C01814=1052.685,226.310,-95.287,172.073,35.922,156.749
C01815=1052.692,226.559,-95.315,172.074,35.926,156.749
C01816=1052.699,226.807,-95.341,172.076,35.929,156.750
C01817=1052.705,227.055,-95.369,172.079,35.932,156.751
C01818=1052.711,227.304,-95.396,172.081,35.936,156.752
C01819=1052.718,227.552,-95.423,172.083,35.939,156.752
C01820=1052.724,227.801,-95.450,172.086,35.942,156.753
C01821=1052.731,228.049,-95.478,172.088,35.946,156.754
C01822=1052.736,228.298,-95.504,172.089,35.950,156.754
C01823=1052.743,228.546,-95.532,172.092,35.953,156.755
C01824=1052.750,228.795,-95.560,172.094,35.956,156.756
C01825=1052.756,229.043,-95.586,172.097,35.960,156.756
C01826=1052.763,229.291,-95.614,172.099,35.963,156.757
C01827=1052.769,229.541,-95.641,172.101,35.966,156.758
C01828=1052.775,229.788,-95.669,172.104,35.970,156.759
C01829=1052.781,230.037,-95.696,172.105,35.974,156.759
C01830=1052.788,230.286,-95.723,172.107,35.977,156.760
C01831=1052.794,230.534,-95.751,172.110,35.980,156.761
C01832=1052.800,230.782,-95.778,172.112,35.984,156.761
C01833=1052.807,231.031,-95.805,172.114,35.987,156.762
C01834=1052.813,231.279,-95.833,172.117,35.990,156.763
C01835=1052.820,231.527,-95.860,172.119,35.994,156.763
C01836=1052.826,231.776,-95.888,172.122,35.997,156.764
C01837=1052.831,232.024,-95.915,172.123,36.001,156.765
C01838=1052.838,232.273,-95.943,172.125,36.004,156.766
C01839=1052.845,232.521,-95.971,172.128,36.008,156.766
C01840=1052.851,232.770,-95.999,172.130,36.011,156.767
C01841=1052.857,233.018,-96.025,172.132,36.015,156.768
C01842=1052.864,233.266,-96.053,172.135,36.018,156.768
C01843=1052.870,233.515,-96.081,172.137,36.021,156.769
C01844=1052.876,233.763,-96.109,172.139,36.025,156.770
C01845=1052.883,234.011,-96.136,172.142,36.028,156.771
C01846=1052.889,234.260,-96.164,172.144,36.031,156.771
C01847=1052.895,234.508,-96.192,172.146,36.035,156.772
C01848=1052.901,234.754,-96.219,172.148,36.039,156.773
C01849=1052.908,235.000,-96.246,172.150,36.042,156.773
C01850=1052.914,235.245,-96.274,172.153,36.045,156.774
C01851=1052.920,235.491,-96.301,172.155,36.049,156.775
C01852=1052.926,235.736,-96.329,172.157,36.052,156.775
C01853=1052.932,235.982,-96.356,172.160,36.055,156.776
C01854=1052.939,236.227,-96.384,172.162,36.059,156.777
C01855=1052.945,236.473,-96.411,172.164,36.062,156.777
C01856=1052.951,236.722,-96.439,172.167,36.065,156.778
C01857=1052.957,236.969,-96.466,172.169,36.069,156.779
C01858=1052.964,237.218,-96.494,172.172,36.072,156.780
C01859=1052.971,237.466,-96.522,172.174,36.076,156.780
C01860=1052.977,237.715,-96.550,172.175,36.079,156.781
C01861=1052.983,237.963,-96.578,172.178,36.082,156.782
C01862=1052.990,238.212,-96.606,172.180,36.086,156.782
C01863=1052.996,238.459,-96.634,172.182,36.089,156.783
C01864=1053.002,238.708,-96.662,172.185,36.093,156.784
C01865=1053.009,238.956,-96.690,172.187,36.096,156.785
C01866=1053.015,239.205,-96.718,172.190,36.099,156.785
C01867=1053.022,239.453,-96.746,172.192,36.103,156.786
C01868=1053.028,239.702,-96.774,172.194,36.106,156.787
C01869=1053.034,239.950,-96.802,172.197,36.109,156.787
C01870=1053.040,240.198,-96.829,172.199,36.113,156.788
C01871=1053.047,240.447,-96.857,172.201,36.116,156.789
C01872=1053.053,240.695,-96.886,172.204,36.120,156.789
C01873=1053.060,240.943,-96.914,172.206,36.123,156.790
C01874=1053.067,241.192,-96.941,172.209,36.126,156.791
C01875=1053.072,241.440,-96.970,172.211,36.130,156.792
C01876=1053.079,241.689,-96.998,172.213,36.133,156.792
C01877=1053.085,241.936,-97.026,172.216,36.136,156.793
C01878=1053.091,242.185,-97.054,172.218,36.140,156.794
C01879=1053.097,242.433,-97.082,172.221,36.143,156.794
C01880=1053.104,242.682,-97.110,172.223,36.147,156.795
C01881=1053.110,242.930,-97.139,172.225,36.150,156.796
C01882=1053.116,243.179,-97.167,172.228,36.154,156.797
C01883=1053.123,243.427,-97.195,172.230,36.157,156.797
C01884=1053.129,243.675,-97.224,172.232,36.161,156.798
C01885=1053.135,243.923,-97.252,172.235,36.164,156.799
C01886=1053.142,244.171,-97.281,172.237,36.167,156.799
C01887=1053.148,244.420,-97.309,172.240,36.171,156.800
C01888=1053.154,244.668,-97.337,172.242,36.174,156.801
C01889=1053.160,244.917,-97.366,172.244,36.177,156.802
C01890=1053.167,245.165,-97.393,172.247,36.181,156.802
C01891=1053.173,245.413,-97.422,172.249,36.184,156.803
C01892=1053.179,245.662,-97.451,172.252,36.187,156.804
C01893=1053.186,245.910,-97.478,172.254,36.191,156.804
C01894=1053.192,246.158,-97.508,172.257,36.195,156.805
C01895=1053.198,246.407,-97.536,172.260,36.198,156.806
C01896=1053.204,246.655,-97.565,172.262,36.202,156.807
C01897=1053.211,246.903,-97.593,172.264,36.205,156.807
C01898=1053.217,247.151,-97.621,172.267,36.208,156.808
C01899=1053.223,247.399,-97.650,172.269,36.212,156.809
C01900=1053.229,247.648,-97.679,172.272,36.215,156.809
C01901=1053.235,247.896,-97.708,172.274,36.219,156.810
C01902=1053.241,248.145,-97.736,172.276,36.222,156.811
C01903=1053.248,248.393,-97.764,172.279,36.225,156.812
C01904=1053.254,248.636,-97.793,172.281,36.229,156.812
C01905=1053.260,248.878,-97.820,172.284,36.232,156.813
C01906=1053.266,249.121,-97.849,172.286,36.235,156.814
C01907=1053.272,249.363,-97.877,172.288,36.239,156.814
C01908=1053.279,249.606,-97.905,172.291,36.242,156.815
C01909=1053.284,249.848,-97.933,172.293,36.245,156.816
C01910=1053.290,250.091,-97.961,172.296,36.249,156.817
C01911=1053.297,250.333,-97.989,172.298,36.252,156.817
C01912=1053.303,250.582,-98.018,172.300,36.256,156.818
C01913=1053.310,250.830,-98.047,172.303,36.259,156.819
C01914=1053.316,251.078,-98.075,172.305,36.263,156.819
C01915=1053.322,251.327,-98.104,172.308,36.266,156.820
C01916=1053.328,251.575,-98.133,172.311,36.269,156.821
C01917=1053.334,251.823,-98.163,172.313,36.273,156.822
C01918=1053.340,252.072,-98.191,172.316,36.276,156.822
C01919=1053.347,252.319,-98.219,172.318,36.280,156.823
C01920=1053.354,252.568,-98.248,172.321,36.283,156.824
C01921=1053.360,252.816,-98.277,172.323,36.286,156.824
C01922=1053.366,253.064,-98.306,172.325,36.290,156.825
C01923=1053.372,253.312,-98.335,172.328,36.293,156.826
C01924=1053.378,253.561,-98.364,172.330,36.296,156.827
C01925=1053.385,253.809,-98.393,172.334,36.300,156.827
C01926=1053.391,254.057,-98.422,172.336,36.304,156.828
C01927=1053.398,254.306,-98.451,172.338,36.306,156.829
C01928=1053.404,254.554,-98.480,172.341,36.310,156.829
C01929=1053.411,254.802,-98.509,172.343,36.314,156.830
C01930=1053.417,255.050,-98.538,172.346,36.317,156.831
C01931=1053.423,255.298,-98.567,172.348,36.320,156.832
C01932=1053.430,255.546,-98.596,172.351,36.324,156.832
C01933=1053.436,255.794,-98.625,172.354,36.327,156.833
C01934=1053.443,256.043,-98.654,172.356,36.330,156.834
C01935=1053.449,256.291,-98.683,172.359,36.334,156.834
C01936=1053.455,256.539,-98.712,172.361,36.337,156.835
C01937=1053.461,256.788,-98.741,172.364,36.341,156.836
C01938=1053.468,257.036,-98.770,172.367,36.344,156.837
C01939=1053.475,257.284,-98.800,172.369,36.347,156.837
C01940=1053.481,257.533,-98.829,172.372,36.351,156.838
C01941=1053.487,257.781,-98.858,172.374,36.354,156.839
C01942=1053.493,258.029,-98.887,172.377,36.357,156.839
C01943=1053.500,258.277,-98.915,172.380,36.361,156.840
C01944=1053.507,258.526,-98.945,172.382,36.364,156.841
C01945=1053.513,258.774,-98.974,172.385,36.367,156.842
C01946=1053.520,259.022,-99.003,172.387,36.371,156.842
C01947=1053.526,259.269,-99.033,172.390,36.374,156.843
C01948=1053.533,259.518,-99.062,172.393,36.377,156.844
C01949=1053.539,259.766,-99.091,172.395,36.381,156.844
C01950=1053.546,260.014,-99.120,172.398,36.384,156.845
C01951=1053.552,260.263,-99.149,172.400,36.387,156.846
C01952=1053.559,260.511,-99.179,172.404,36.391,156.847
C01953=1053.565,260.759,-99.208,172.406,36.394,156.847
C01954=1053.571,261.007,-99.237,172.408,36.397,156.848
C01955=1053.578,261.256,-99.267,172.411,36.401,156.849
C01956=1053.585,261.504,-99.296,172.414,36.404,156.849
C01957=1053.591,261.751,-99.326,172.417,36.407,156.850
C01958=1053.598,262.000,-99.355,172.419,36.411,156.851
C01959=1053.604,262.248,-99.384,172.422,36.414,156.852
C01960=1053.610,262.490,-99.413,172.424,36.417,156.852
C01961=1053.617,262.732,-99.442,172.427,36.421,156.853
C01962=1053.623,262.973,-99.470,172.430,36.424,156.854
C01963=1053.629,263.215,-99.499,172.432,36.427,156.854
C01964=1053.635,263.457,-99.528,172.435,36.430,156.855
C01965=1053.642,263.699,-99.557,172.437,36.434,156.856
C01966=1053.648,263.940,-99.585,172.440,36.437,156.856
C01967=1053.654,264.181,-99.614,172.443,36.440,156.857
C01968=1053.660,264.429,-99.644,172.445,36.444,156.858
C01969=1053.667,264.678,-99.674,172.448,36.447,156.859
C01970=1053.674,264.925,-99.703,172.451,36.451,156.859
C01971=1053.679,265.174,-99.733,172.454,36.454,156.860
C01972=1053.686,265.422,-99.763,172.456,36.458,156.861
C01973=1053.692,265.670,-99.792,172.458,36.461,156.862
C01974=1053.698,265.918,-99.823,172.462,36.464,156.862
C01975=1053.705,266.167,-99.852,172.464,36.468,156.863
C01976=1053.712,266.414,-99.882,172.467,36.472,156.864
C01977=1053.717,266.662,-99.912,172.469,36.475,156.865
C01978=1053.724,266.911,-99.941,172.473,36.478,156.865
C01979=1053.731,267.159,-99.971,172.475,36.482,156.866
C01980=1053.736,267.407,-100.001,172.477,36.485,156.867
C01981=1053.744,267.655,-100.031,172.481,36.489,156.867
C01982=1053.750,267.903,-100.061,172.483,36.492,156.868
C01983=1053.756,268.152,-100.091,172.486,36.495,156.869
C01984=1053.763,268.399,-100.121,172.489,36.499,156.870
C01985=1053.769,268.647,-100.151,172.492,36.502,156.870
C01986=1053.775,268.896,-100.180,172.494,36.506,156.871
C01987=1053.781,269.144,-100.211,172.498,36.509,156.872
C01988=1053.788,269.392,-100.241,172.500,36.513,156.873
C01989=1053.794,269.640,-100.271,172.502,36.516,156.873
C01990=1053.801,269.889,-100.301,172.505,36.519,156.874
C01991=1053.807,270.137,-100.331,172.508,36.523,156.875
C01992=1053.813,270.384,-100.361,172.511,36.526,156.876
C01993=1053.820,270.633,-100.391,172.513,36.530,156.876
C01994=1053.826,270.880,-100.421,172.517,36.533,156.877
C01995=1053.833,271.129,-100.452,172.519,36.537,156.878
C01996=1053.839,271.377,-100.481,172.522,36.540,156.879
C01997=1053.846,271.625,-100.512,172.525,36.543,156.879
C01998=1053.852,271.873,-100.541,172.527,36.547,156.880
C01999=1053.858,272.121,-100.572,172.531,36.550,156.881
C02000=1053.865,272.369,-100.602,172.533,36.554,156.882
C02001=1053.871,272.617,-100.633,172.536,36.557,156.882
C02002=1053.877,272.865,-100.663,172.539,36.561,156.883
C02003=1053.884,273.113,-100.693,172.542,36.564,156.884
C02004=1053.890,273.361,-100.723,172.544,36.568,156.885
C02005=1053.897,273.610,-100.754,172.548,36.571,156.885
C02006=1053.903,273.857,-100.784,172.550,36.575,156.886
C02007=1053.910,274.106,-100.815,172.552,36.578,156.887
C02008=1053.915,274.354,-100.845,172.556,36.581,156.887
C02009=1053.923,274.602,-100.875,172.558,36.585,156.888
C02010=1053.928,274.850,-100.905,172.562,36.588,156.889
C02011=1053.935,275.098,-100.936,172.564,36.592,156.890
C02012=1053.941,275.346,-100.966,172.567,36.595,156.891
C02013=1053.948,275.594,-100.997,172.570,36.599,156.891
C02014=1053.954,275.842,-101.027,172.573,36.602,156.892
C02015=1053.960,276.091,-101.058,172.575,36.606,156.893
C02016=1053.966,276.334,-101.088,172.579,36.609,156.894
C02017=1053.973,276.577,-101.118,172.581,36.613,156.894
C02018=1053.979,276.821,-101.148,172.584,36.616,156.895
C02019=1053.985,277.064,-101.178,172.587,36.619,156.896
C02020=1053.992,277.308,-101.208,172.589,36.623,156.896
C02021=1053.999,277.552,-101.238,172.593,36.626,156.897
C02022=1054.004,277.796,-101.268,172.595,36.630,156.898
C02023=1054.010,278.039,-101.298,172.598,36.633,156.899
C02024=1054.018,278.287,-101.328,172.601,36.637,156.900
C02025=1054.023,278.535,-101.359,172.604,36.640,156.900
C02026=1054.030,278.783,-101.390,172.607,36.643,156.901
C02027=1054.036,279.031,-101.421,172.610,36.647,156.902
C02028=1054.042,279.279,-101.451,172.613,36.650,156.902
C02029=1054.050,279.527,-101.482,172.616,36.654,156.903
C02030=1054.056,279.775,-101.513,172.619,36.657,156.904
C02031=1054.062,280.023,-101.543,172.621,36.661,156.905
C02032=1054.069,280.271,-101.574,172.624,36.664,156.906
C02033=1054.075,280.519,-101.605,172.627,36.668,156.906
C02034=1054.081,280.767,-101.636,172.630,36.672,156.907
C02035=1054.088,281.015,-101.667,172.633,36.675,156.908
C02036=1054.094,281.262,-101.698,172.636,36.679,156.909
C02037=1054.100,281.511,-101.729,172.639,36.682,156.909
C02038=1054.107,281.759,-101.759,172.642,36.686,156.910
C02039=1054.113,282.007,-101.790,172.645,36.689,156.911
C02040=1054.120,282.255,-101.822,172.648,36.693,156.912
C02041=1054.126,282.503,-101.853,172.650,36.696,156.913
C02042=1054.132,282.750,-101.884,172.654,36.700,156.913
C02043=1054.138,282.999,-101.914,172.656,36.703,156.914
C02044=1054.145,283.247,-101.946,172.660,36.707,156.915
C02045=1054.152,283.495,-101.977,172.662,36.710,156.916
C02046=1054.158,283.742,-102.008,172.666,36.714,156.916
C02047=1054.164,283.990,-102.039,172.668,36.717,156.917
C02048=1054.171,284.239,-102.070,172.672,36.721,156.918
C02049=1054.177,284.486,-102.101,172.674,36.724,156.919
C02050=1054.183,284.735,-102.132,172.678,36.728,156.919
C02051=1054.189,284.983,-102.164,172.680,36.732,156.920
C02052=1054.196,285.231,-102.195,172.684,36.735,156.921
C02053=1054.203,285.479,-102.226,172.686,36.739,156.922
C02054=1054.209,285.726,-102.257,172.690,36.742,156.923
C02055=1054.215,285.974,-102.288,172.693,36.746,156.923
C02056=1054.222,286.222,-102.320,172.696,36.749,156.924
C02057=1054.229,286.471,-102.350,172.699,36.753,156.925
C02058=1054.235,286.719,-102.382,172.702,36.756,156.926
C02059=1054.241,286.966,-102.413,172.705,36.760,156.926
C02060=1054.248,287.214,-102.444,172.708,36.763,156.927
C02061=1054.255,287.462,-102.476,172.711,36.766,156.928
C02062=1054.261,287.710,-102.506,172.714,36.770,156.929
C02063=1054.268,287.958,-102.538,172.717,36.773,156.930
C02064=1054.275,288.206,-102.569,172.720,36.778,156.930
C02065=1054.280,288.453,-102.601,172.723,36.781,156.931
C02066=1054.287,288.701,-102.632,172.727,36.784,156.932
C02067=1054.294,288.949,-102.664,172.729,36.788,156.933
C02068=1054.300,289.197,-102.695,172.733,36.791,156.934
C02069=1054.306,289.445,-102.727,172.735,36.795,156.934
C02070=1054.313,289.693,-102.759,172.739,36.799,156.935
C02071=1054.319,289.941,-102.790,172.741,36.802,156.936
C02072=1054.326,290.191,-102.821,172.745,36.806,156.937
C02073=1054.332,290.442,-102.854,172.748,36.809,156.938
C02074=1054.339,290.692,-102.886,172.751,36.813,156.938
C02075=1054.345,290.943,-102.917,172.754,36.817,156.939
C02076=1054.352,291.190,-102.949,172.757,36.820,156.940
C02077=1054.358,291.439,-102.981,172.760,36.824,156.941
C02078=1054.364,291.686,-103.012,172.764,36.828,156.942
C02079=1054.371,291.934,-103.044,172.766,36.831,156.942
C02080=1054.377,292.182,-103.076,172.770,36.835,156.943
C02081=1054.384,292.430,-103.107,172.772,36.838,156.944
C02082=1054.390,292.678,-103.139,172.776,36.842,156.945
C02083=1054.397,292.926,-103.171,172.779,36.846,156.946
C02084=1054.404,293.173,-103.203,172.782,36.849,156.946
C02085=1054.410,293.421,-103.235,172.785,36.853,156.947
C02086=1054.416,293.669,-103.266,172.788,36.856,156.948
C02087=1054.423,293.917,-103.298,172.791,36.860,156.949
C02088=1054.429,294.165,-103.331,172.795,36.864,156.950
C02089=1054.436,294.413,-103.362,172.797,36.867,156.950
C02090=1054.442,294.661,-103.394,172.801,36.871,156.951
C02091=1054.449,294.909,-103.425,172.804,36.875,156.952
C02092=1054.456,295.156,-103.458,172.807,36.878,156.953
C02093=1054.462,295.404,-103.490,172.810,36.882,156.954
C02094=1054.468,295.652,-103.521,172.814,36.886,156.955
C02095=1054.475,295.900,-103.554,172.817,36.889,156.955
C02096=1054.482,296.148,-103.585,172.820,36.893,156.956
C02097=1054.488,296.395,-103.618,172.824,36.897,156.957
C02098=1054.494,296.644,-103.650,172.826,36.900,156.958
C02099=1054.501,296.891,-103.682,172.830,36.904,156.959
C02100=1054.507,297.139,-103.714,172.832,36.908,156.959
C02101=1054.513,297.387,-103.747,172.836,36.912,156.960
C02102=1054.519,297.635,-103.779,172.839,36.915,156.961
C02103=1054.526,297.882,-103.811,172.842,36.919,156.962
C02104=1054.532,298.130,-103.843,172.845,36.923,156.963
C02105=1054.538,298.378,-103.876,172.849,36.927,156.964
C02106=1054.544,298.626,-103.908,172.852,36.930,156.964
C02107=1054.551,298.874,-103.941,172.855,36.934,156.965
C02108=1054.558,299.121,-103.973,172.859,36.938,156.966
C02109=1054.564,299.369,-104.005,172.861,36.942,156.967
C02110=1054.570,299.617,-104.038,172.865,36.945,156.968
C02111=1054.576,299.864,-104.070,172.868,36.949,156.969
C02112=1054.582,300.113,-104.102,172.872,36.953,156.970
C02113=1054.589,300.360,-104.134,172.874,36.957,156.970
C02114=1054.596,300.608,-104.167,172.878,36.960,156.971
C02115=1054.602,300.856,-104.199,172.882,36.964,156.972
C02116=1054.608,301.103,-104.232,172.884,36.968,156.973
C02117=1054.614,301.351,-104.265,172.888,36.972,156.974
C02118=1054.621,301.598,-104.297,172.891,36.975,156.975
C02119=1054.627,301.846,-104.329,172.894,36.979,156.976
C02120=1054.634,302.095,-104.362,172.897,36.983,156.976
C02121=1054.640,302.342,-104.395,172.901,36.987,156.977
C02122=1054.647,302.590,-104.427,172.904,36.990,156.978
C02123=1054.654,302.837,-104.460,172.907,36.994,156.979
C02124=1054.660,303.085,-104.492,172.911,36.997,156.980
C02125=1054.666,303.332,-104.525,172.914,37.001,156.981
C02126=1054.672,303.581,-104.557,172.918,37.005,156.981
C02127=1054.679,303.829,-104.590,172.920,37.009,156.982
C02128=1054.686,304.095,-104.625,172.924,37.013,156.983
C02129=1054.694,304.361,-104.660,172.928,37.017,156.984
C02130=1054.700,304.627,-104.695,172.931,37.021,156.985
C02131=1054.707,304.894,-104.731,172.935,37.025,156.986
C02132=1054.713,305.141,-104.763,172.938,37.029,156.987
C02133=1054.720,305.389,-104.796,172.942,37.033,156.988
C02134=1054.727,305.637,-104.829,172.945,37.036,156.989
C02135=1054.733,305.885,-104.862,172.948,37.041,156.989
C02136=1054.740,306.132,-104.894,172.952,37.044,156.990
C02137=1054.746,306.380,-104.927,172.955,37.048,156.991
C02138=1054.753,306.628,-104.960,172.959,37.052,156.992
C02139=1054.759,306.875,-104.993,172.962,37.055,156.993
C02140=1054.766,307.122,-105.026,172.966,37.059,156.994
C02141=1054.773,307.371,-105.059,172.969,37.063,156.995
C02142=1054.779,307.618,-105.092,172.972,37.067,156.995
C02143=1054.785,307.866,-105.125,172.976,37.071,156.996
C02144=1054.793,308.114,-105.157,172.979,37.074,156.997
C02145=1054.799,308.361,-105.190,172.983,37.078,156.998
C02146=1054.806,308.608,-105.223,172.987,37.082,156.999
C02147=1054.813,308.857,-105.257,172.989,37.086,157.000
C02148=1054.819,309.104,-105.289,172.993,37.090,157.001
C02149=1054.825,309.352,-105.322,172.996,37.094,157.002
C02150=1054.833,309.600,-105.356,173.000,37.097,157.002
C02151=1054.839,309.847,-105.389,173.003,37.101,157.003
C02152=1054.846,310.095,-105.422,173.007,37.105,157.004
C02153=1054.852,310.343,-105.454,173.011,37.109,157.005
C02154=1054.859,310.591,-105.488,173.013,37.113,157.006
C02155=1054.866,310.838,-105.521,173.017,37.117,157.007
C02156=1054.873,311.086,-105.553,173.020,37.120,157.008
C02157=1054.880,311.333,-105.587,173.024,37.124,157.008
C02158=1054.886,311.581,-105.620,173.028,37.128,157.009
C02159=1054.893,311.829,-105.654,173.031,37.131,157.010
C02160=1054.900,312.076,-105.686,173.035,37.135,157.011
C02161=1054.907,312.324,-105.719,173.038,37.139,157.012
C02162=1054.913,312.571,-105.753,173.042,37.143,157.013
C02163=1054.920,312.820,-105.786,173.045,37.147,157.014
C02164=1054.927,313.067,-105.819,173.048,37.151,157.015
C02165=1054.934,313.315,-105.853,173.052,37.155,157.016
C02166=1054.940,313.562,-105.886,173.055,37.159,157.016
C02167=1054.946,313.811,-105.920,173.059,37.163,157.017
C02168=1054.953,314.057,-105.953,173.063,37.167,157.018
C02169=1054.959,314.305,-105.988,173.066,37.171,157.019
C02170=1054.966,314.553,-106.020,173.070,37.175,157.020
C02171=1054.972,314.801,-106.055,173.074,37.179,157.021
C02172=1054.979,315.048,-106.088,173.076,37.183,157.022
C02173=1054.985,315.295,-106.122,173.080,37.187,157.023
C02174=1054.991,315.544,-106.155,173.084,37.191,157.024
C02175=1054.997,315.791,-106.189,173.087,37.195,157.025
C02176=1055.005,316.039,-106.223,173.091,37.199,157.026
C02177=1055.010,316.286,-106.257,173.094,37.203,157.027
C02178=1055.017,316.534,-106.290,173.098,37.207,157.028
C02179=1055.023,316.781,-106.324,173.102,37.211,157.028
C02180=1055.030,317.029,-106.358,173.105,37.215,157.029
C02181=1055.036,317.276,-106.392,173.109,37.219,157.030
C02182=1055.043,317.524,-106.426,173.113,37.223,157.031
C02183=1055.050,317.772,-106.461,173.116,37.227,157.032
C02184=1055.057,318.042,-106.497,173.120,37.231,157.033
C02185=1055.064,318.312,-106.534,173.124,37.236,157.034
C02186=1055.072,318.583,-106.571,173.128,37.240,157.035
C02187=1055.079,318.853,-106.608,173.131,37.245,157.036
C02188=1055.085,319.101,-106.643,173.135,37.249,157.037
C02189=1055.091,319.349,-106.677,173.139,37.253,157.038
C02190=1055.098,319.596,-106.711,173.142,37.257,157.039
C02191=1055.105,319.844,-106.745,173.146,37.261,157.040
C02192=1055.111,320.091,-106.778,173.149,37.265,157.041
C02193=1055.118,320.339,-106.813,173.153,37.269,157.042
C02194=1055.125,320.587,-106.847,173.157,37.273,157.043
C02195=1055.131,320.834,-106.881,173.161,37.277,157.044
C02196=1055.138,321.082,-106.915,173.164,37.281,157.045
C02197=1055.144,321.330,-106.949,173.168,37.285,157.046
C02198=1055.151,321.577,-106.982,173.172,37.290,157.047
C02199=1055.157,321.825,-107.017,173.175,37.294,157.048
C02200=1055.164,322.073,-107.051,173.179,37.298,157.049
C02201=1055.171,322.320,-107.086,173.183,37.302,157.050
C02202=1055.177,322.567,-107.120,173.186,37.305,157.050
C02203=1055.185,322.815,-107.154,173.190,37.310,157.052
C02204=1055.191,323.063,-107.188,173.194,37.314,157.052
C02205=1055.197,323.311,-107.223,173.198,37.318,157.053
C02206=1055.205,323.558,-107.257,173.202,37.322,157.054
C02207=1055.211,323.805,-107.291,173.206,37.326,157.055
C02208=1055.218,324.053,-107.325,173.209,37.330,157.056
C02209=1055.225,324.300,-107.360,173.213,37.334,157.057
C02210=1055.231,324.548,-107.395,173.217,37.339,157.058
C02211=1055.238,324.796,-107.428,173.220,37.343,157.059
C02212=1055.245,325.042,-107.463,173.224,37.347,157.060
C02213=1055.252,325.290,-107.497,173.228,37.351,157.061
C02214=1055.258,325.538,-107.531,173.231,37.355,157.062
C02215=1055.265,325.785,-107.567,173.235,37.359,157.063
C02216=1055.272,326.033,-107.600,173.239,37.364,157.064
C02217=1055.279,326.281,-107.635,173.243,37.368,157.065
C02218=1055.285,326.529,-107.670,173.246,37.372,157.066
C02219=1055.293,326.776,-107.704,173.251,37.376,157.067
C02220=1055.299,327.024,-107.739,173.255,37.380,157.068
C02221=1055.307,327.271,-107.773,173.258,37.384,157.069
C02222=1055.313,327.519,-107.808,173.262,37.389,157.070
C02223=1055.320,327.766,-107.843,173.266,37.393,157.071
C02224=1055.327,328.013,-107.876,173.270,37.397,157.072
C02225=1055.334,328.260,-107.912,173.273,37.401,157.073
C02226=1055.340,328.508,-107.946,173.277,37.405,157.074
C02227=1055.347,328.755,-107.980,173.282,37.409,157.075
C02228=1055.354,329.003,-108.016,173.285,37.413,157.076
C02229=1055.361,329.251,-108.050,173.289,37.418,157.077
C02230=1055.369,329.498,-108.085,173.293,37.422,157.078
C02231=1055.376,329.746,-108.120,173.297,37.426,157.079
C02232=1055.382,329.994,-108.155,173.300,37.430,157.080
C02233=1055.389,330.241,-108.190,173.305,37.435,157.081
C02234=1055.396,330.489,-108.225,173.309,37.439,157.082
C02235=1055.402,330.736,-108.260,173.312,37.443,157.083
C02236=1055.409,330.984,-108.294,173.316,37.448,157.084
C02237=1055.416,331.231,-108.329,173.320,37.452,157.085
C02238=1055.422,331.479,-108.365,173.324,37.456,157.086
C02239=1055.429,331.726,-108.400,173.328,37.461,157.087
C02240=1055.436,331.991,-108.438,173.332,37.465,157.088
C02241=1055.444,332.255,-108.475,173.336,37.470,157.089
C02242=1055.451,332.521,-108.512,173.341,37.475,157.090
C02243=1055.458,332.786,-108.550,173.345,37.479,157.091
C02244=1055.465,333.034,-108.585,173.348,37.484,157.092
C02245=1055.471,333.281,-108.620,173.353,37.488,157.094
C02246=1055.478,333.528,-108.655,173.357,37.492,157.094
C02247=1055.485,333.776,-108.691,173.361,37.497,157.096
C02248=1055.492,334.024,-108.726,173.364,37.501,157.097
C02249=1055.499,334.271,-108.761,173.368,37.506,157.098
C02250=1055.505,334.519,-108.797,173.373,37.510,157.099
C02251=1055.512,334.766,-108.833,173.377,37.514,157.100
C02252=1055.519,335.013,-108.868,173.381,37.519,157.101
C02253=1055.526,335.260,-108.903,173.384,37.523,157.102
C02254=1055.532,335.508,-108.938,173.389,37.527,157.103
C02255=1055.540,335.756,-108.974,173.393,37.532,157.104
C02256=1055.547,336.003,-109.009,173.397,37.536,157.105
C02257=1055.554,336.250,-109.045,173.400,37.541,157.106
C02258=1055.560,336.497,-109.080,173.405,37.545,157.107
C02259=1055.566,336.745,-109.116,173.409,37.550,157.108
C02260=1055.574,336.993,-109.151,173.413,37.554,157.109
C02261=1055.581,337.240,-109.187,173.417,37.559,157.110
C02262=1055.587,337.487,-109.223,173.421,37.563,157.111
C02263=1055.594,337.734,-109.258,173.425,37.568,157.113
C02264=1055.601,337.982,-109.294,173.429,37.572,157.114
C02265=1055.608,338.230,-109.329,173.433,37.577,157.115
C02266=1055.614,338.477,-109.366,173.438,37.581,157.116
C02267=1055.621,338.724,-109.401,173.441,37.586,157.117
C02268=1055.628,338.971,-109.437,173.445,37.590,157.118
C02269=1055.635,339.219,-109.473,173.450,37.595,157.119
C02270=1055.642,339.466,-109.509,173.454,37.600,157.120
C02271=1055.649,339.713,-109.544,173.458,37.604,157.121
C02272=1055.656,339.961,-109.580,173.463,37.609,157.122
C02273=1055.662,340.208,-109.616,173.466,37.613,157.123
C02274=1055.669,340.455,-109.652,173.470,37.618,157.125
C02275=1055.676,340.702,-109.688,173.474,37.622,157.126
C02276=1055.683,340.950,-109.723,173.479,37.627,157.127
C02277=1055.690,341.197,-109.760,173.483,37.632,157.128
C02278=1055.697,341.445,-109.795,173.487,37.636,157.129
C02279=1055.704,341.692,-109.831,173.491,37.640,157.130
C02280=1055.710,341.939,-109.868,173.495,37.646,157.131
C02281=1055.718,342.187,-109.904,173.500,37.650,157.132
C02282=1055.724,342.434,-109.940,173.504,37.654,157.133
C02283=1055.731,342.681,-109.975,173.508,37.659,157.135
C02284=1055.739,342.928,-110.012,173.513,37.664,157.136
C02285=1055.745,343.176,-110.048,173.516,37.668,157.137
C02286=1055.753,343.424,-110.084,173.520,37.673,157.138
C02287=1055.759,343.671,-110.120,173.525,37.678,157.139
C02288=1055.766,343.918,-110.157,173.529,37.682,157.140
C02289=1055.773,344.165,-110.193,173.534,37.687,157.141
C02290=1055.779,344.412,-110.229,173.538,37.692,157.142
C02291=1055.787,344.660,-110.265,173.542,37.697,157.144
C02292=1055.793,344.907,-110.302,173.546,37.701,157.145
C02293=1055.800,345.154,-110.339,173.550,37.706,157.146
C02294=1055.807,345.401,-110.374,173.555,37.711,157.147
C02295=1055.814,345.649,-110.411,173.559,37.716,157.148
C02296=1055.821,345.910,-110.450,173.564,37.721,157.150
C02297=1055.828,346.171,-110.488,173.568,37.726,157.151
C02298=1055.835,346.432,-110.527,173.573,37.731,157.152
C02299=1055.844,346.693,-110.565,173.577,37.736,157.153
C02300=1055.850,346.940,-110.601,173.582,37.741,157.154
C02301=1055.857,347.188,-110.638,173.586,37.745,157.155
C02302=1055.865,347.434,-110.675,173.591,37.750,157.157
C02303=1055.871,347.681,-110.711,173.594,37.755,157.158
C02304=1055.878,347.928,-110.748,173.599,37.760,157.159
C02305=1055.885,348.176,-110.785,173.603,37.765,157.160
C02306=1055.893,348.423,-110.822,173.608,37.770,157.161
C02307=1055.899,348.670,-110.858,173.612,37.775,157.163
C02308=1055.906,348.918,-110.895,173.617,37.779,157.164
C02309=1055.912,349.165,-110.931,173.621,37.784,157.165
C02310=1055.920,349.412,-110.968,173.626,37.789,157.166
C02311=1055.927,349.660,-111.005,173.630,37.794,157.167
C02312=1055.934,349.906,-111.042,173.635,37.799,157.169
C02313=1055.941,350.154,-111.079,173.639,37.803,157.170
C02314=1055.948,350.401,-111.115,173.643,37.808,157.171
C02315=1055.955,350.648,-111.152,173.647,37.813,157.172
C02316=1055.962,350.895,-111.189,173.652,37.818,157.173
C02317=1055.969,351.142,-111.227,173.656,37.823,157.175
C02318=1055.976,351.390,-111.263,173.661,37.828,157.176
C02319=1055.984,351.636,-111.300,173.665,37.833,157.177
C02320=1055.991,351.884,-111.337,173.670,37.838,157.178
C02321=1055.997,352.131,-111.374,173.674,37.843,157.180
C02322=1056.004,352.378,-111.412,173.679,37.848,157.181
C02323=1056.011,352.625,-111.448,173.683,37.853,157.182
C02324=1056.018,352.872,-111.486,173.688,37.858,157.183
C02325=1056.025,353.119,-111.523,173.692,37.863,157.184
C02326=1056.032,353.367,-111.560,173.697,37.868,157.186
C02327=1056.039,353.614,-111.597,173.702,37.873,157.187
C02328=1056.046,353.860,-111.635,173.706,37.879,157.188
C02329=1056.053,354.107,-111.672,173.711,37.884,157.189
C02330=1056.060,354.355,-111.709,173.715,37.889,157.191
C02331=1056.068,354.602,-111.747,173.720,37.894,157.192
C02332=1056.075,354.850,-111.784,173.724,37.899,157.193
C02333=1056.081,355.096,-111.821,173.729,37.904,157.195
C02334=1056.089,355.343,-111.859,173.734,37.909,157.196
C02335=1056.096,355.590,-111.896,173.738,37.914,157.197
C02336=1056.103,355.837,-111.934,173.743,37.919,157.198
C02337=1056.110,356.084,-111.971,173.747,37.925,157.200
C02338=1056.118,356.332,-112.009,173.752,37.929,157.201
C02339=1056.125,356.579,-112.046,173.757,37.934,157.202
C02340=1056.132,356.825,-112.084,173.761,37.940,157.203
C02341=1056.139,357.072,-112.121,173.766,37.945,157.205
C02342=1056.146,357.319,-112.159,173.771,37.950,157.206
C02343=1056.153,357.567,-112.196,173.775,37.955,157.207
C02344=1056.160,357.814,-112.234,173.780,37.960,157.208
C02345=1056.167,358.061,-112.272,173.785,37.966,157.210
C02346=1056.174,358.308,-112.309,173.789,37.971,157.211
C02347=1056.181,358.555,-112.347,173.794,37.976,157.212
C02348=1056.189,358.802,-112.385,173.799,37.981,157.214
C02349=1056.196,359.049,-112.423,173.803,37.987,157.215
C02350=1056.203,359.297,-112.461,173.808,37.992,157.216
C02351=1056.210,359.544,-112.498,173.813,37.997,157.218
C02352=1056.217,359.809,-112.539,173.818,38.003,157.219
C02353=1056.225,360.075,-112.580,173.823,38.009,157.221
C02354=1056.233,360.341,-112.621,173.829,38.014,157.222
C02355=1056.241,360.607,-112.661,173.834,38.020,157.223
C02356=1056.248,360.853,-112.700,173.838,38.025,157.225
C02357=1056.255,361.101,-112.738,173.843,38.031,157.226
C02358=1056.262,361.347,-112.776,173.848,38.036,157.227
C02359=1056.270,361.595,-112.813,173.853,38.041,157.229
C02360=1056.277,361.841,-112.852,173.857,38.047,157.230
C02361=1056.284,362.088,-112.890,173.862,38.052,157.231
C02362=1056.291,362.335,-112.928,173.867,38.058,157.233
C02363=1056.299,362.583,-112.966,173.872,38.063,157.234
C02364=1056.306,362.830,-113.005,173.876,38.068,157.235
C02365=1056.313,363.077,-113.042,173.882,38.073,157.237
C02366=1056.321,363.323,-113.081,173.887,38.079,157.238
C02367=1056.328,363.570,-113.119,173.892,38.084,157.240
C02368=1056.335,363.817,-113.157,173.896,38.090,157.241
C02369=1056.342,364.064,-113.196,173.901,38.095,157.242
C02370=1056.349,364.311,-113.234,173.906,38.101,157.244
C02371=1056.356,364.557,-113.273,173.911,38.106,157.245
C02372=1056.364,364.805,-113.311,173.916,38.112,157.247
C02373=1056.371,365.052,-113.350,173.921,38.118,157.248
C02374=1056.378,365.299,-113.388,173.926,38.123,157.249
C02375=1056.385,365.545,-113.427,173.931,38.129,157.251
C02376=1056.392,365.792,-113.466,173.936,38.134,157.252
C02377=1056.399,366.039,-113.504,173.941,38.140,157.254
C02378=1056.407,366.286,-113.543,173.945,38.146,157.255
C02379=1056.414,366.533,-113.581,173.950,38.151,157.256
C02380=1056.421,366.780,-113.620,173.956,38.157,157.258
C02381=1056.428,367.026,-113.659,173.961,38.163,157.259
C02382=1056.436,367.274,-113.697,173.966,38.168,157.261
C02383=1056.443,367.520,-113.736,173.971,38.173,157.262
C02384=1056.450,367.767,-113.775,173.975,38.180,157.264
C02385=1056.457,368.014,-113.813,173.980,38.185,157.265
C02386=1056.465,368.261,-113.853,173.986,38.190,157.266
C02387=1056.472,368.508,-113.891,173.991,38.196,157.268
C02388=1056.479,368.754,-113.930,173.996,38.202,157.269
C02389=1056.487,369.001,-113.969,174.001,38.208,157.271
C02390=1056.494,369.248,-114.008,174.006,38.213,157.272
C02391=1056.502,369.496,-114.047,174.012,38.219,157.274
C02392=1056.509,369.742,-114.085,174.017,38.225,157.275
C02393=1056.516,369.988,-114.125,174.022,38.231,157.277
C02394=1056.524,370.236,-114.163,174.026,38.236,157.278
C02395=1056.531,370.482,-114.202,174.031,38.242,157.280
C02396=1056.539,370.729,-114.242,174.037,38.248,157.281
C02397=1056.547,370.976,-114.280,174.042,38.254,157.282
C02398=1056.554,371.222,-114.320,174.047,38.260,157.284
C02399=1056.561,371.470,-114.359,174.052,38.266,157.286
C02400=1056.569,371.716,-114.397,174.058,38.271,157.287
C02401=1056.576,371.963,-114.437,174.063,38.277,157.288
C02402=1056.583,372.210,-114.476,174.068,38.283,157.290
C02403=1056.591,372.457,-114.516,174.073,38.289,157.292
C02404=1056.598,372.703,-114.556,174.079,38.295,157.293
C02405=1056.605,372.950,-114.595,174.084,38.301,157.295
C02406=1056.613,373.197,-114.634,174.089,38.307,157.296
C02407=1056.620,373.444,-114.674,174.095,38.313,157.298
C02408=1056.629,373.728,-114.719,174.101,38.319,157.299
C02409=1056.637,374.012,-114.765,174.106,38.326,157.301
C02410=1056.646,374.296,-114.810,174.113,38.333,157.303
C02411=1056.655,374.581,-114.856,174.120,38.340,157.305
C02412=1056.662,374.827,-114.896,174.125,38.346,157.306
C02413=1056.669,375.075,-114.935,174.130,38.352,157.308
C02414=1056.676,375.321,-114.975,174.135,38.358,157.309
C02415=1056.684,375.568,-115.015,174.141,38.364,157.311
C02416=1056.692,375.815,-115.055,174.146,38.370,157.312
C02417=1056.699,376.061,-115.094,174.151,38.377,157.314
C02418=1056.707,376.308,-115.134,174.157,38.383,157.316
C02419=1056.714,376.555,-115.174,174.162,38.389,157.317
C02420=1056.721,376.801,-115.213,174.167,38.395,157.319
C02421=1056.729,377.048,-115.253,174.173,38.401,157.320
C02422=1056.737,377.295,-115.293,174.178,38.407,157.322
C02423=1056.744,377.541,-115.333,174.183,38.414,157.324
C02424=1056.752,377.788,-115.373,174.189,38.420,157.325
C02425=1056.760,378.034,-115.413,174.195,38.426,157.327
C02426=1056.767,378.280,-115.453,174.201,38.432,157.328
C02427=1056.775,378.527,-115.493,174.206,38.438,157.330
C02428=1056.782,378.774,-115.533,174.211,38.444,157.332
C02429=1056.790,379.021,-115.573,174.217,38.451,157.333
C02430=1056.797,379.267,-115.613,174.222,38.457,157.335
C02431=1056.805,379.514,-115.653,174.227,38.463,157.337
C02432=1056.813,379.761,-115.693,174.234,38.469,157.338
C02433=1056.821,380.007,-115.733,174.239,38.476,157.340
C02434=1056.829,380.254,-115.773,174.245,38.482,157.342
C02435=1056.836,380.501,-115.813,174.250,38.488,157.343
C02436=1056.844,380.747,-115.855,174.255,38.495,157.345
C02437=1056.851,380.993,-115.894,174.261,38.501,157.346
C02438=1056.859,381.240,-115.935,174.267,38.507,157.348
C02439=1056.866,381.487,-115.975,174.273,38.514,157.350
C02440=1056.874,381.733,-116.016,174.278,38.520,157.352
C02441=1056.882,381.980,-116.056,174.284,38.527,157.353
C02442=1056.889,382.227,-116.097,174.289,38.533,157.355
C02443=1056.896,382.472,-116.137,174.296,38.540,157.357
C02444=1056.904,382.719,-116.179,174.301,38.546,157.358
C02445=1056.911,382.966,-116.218,174.307,38.553,157.360
C02446=1056.919,383.212,-116.259,174.312,38.559,157.362
C02447=1056.927,383.459,-116.300,174.319,38.566,157.364
C02448=1056.935,383.705,-116.341,174.324,38.573,157.365
C02449=1056.943,383.951,-116.382,174.330,38.579,157.367
C02450=1056.950,384.198,-116.423,174.335,38.585,157.369
C02451=1056.958,384.445,-116.463,174.342,38.592,157.370
C02452=1056.965,384.691,-116.504,174.347,38.599,157.372
C02453=1056.973,384.938,-116.545,174.353,38.605,157.374
C02454=1056.981,385.184,-116.585,174.359,38.612,157.376
C02455=1056.988,385.431,-116.626,174.365,38.619,157.377
C02456=1056.996,385.677,-116.667,174.370,38.625,157.379
C02457=1057.004,385.923,-116.708,174.377,38.632,157.381
C02458=1057.012,386.170,-116.749,174.382,38.639,157.383
C02459=1057.020,386.416,-116.790,174.388,38.646,157.384
C02460=1057.027,386.662,-116.832,174.394,38.652,157.386
C02461=1057.036,386.909,-116.873,174.400,38.659,157.388
C02462=1057.043,387.156,-116.914,174.405,38.665,157.390
C02463=1057.051,387.402,-116.954,174.412,38.672,157.392
C02464=1057.061,387.717,-117.008,174.419,38.681,157.394
C02465=1057.071,388.034,-117.060,174.427,38.690,157.396
C02466=1057.082,388.350,-117.113,174.435,38.698,157.399
C02467=1057.092,388.667,-117.166,174.442,38.707,157.401
C02468=1057.100,388.912,-117.207,174.449,38.714,157.403
C02469=1057.107,389.159,-117.248,174.455,38.721,157.404
C02470=1057.116,389.404,-117.290,174.461,38.728,157.406
C02471=1057.124,389.652,-117.331,174.467,38.735,157.408
C02472=1057.132,389.897,-117.373,174.473,38.742,157.410
C02473=1057.139,390.144,-117.414,174.479,38.749,157.412
C02474=1057.147,390.390,-117.456,174.486,38.756,157.414
C02475=1057.155,390.637,-117.497,174.491,38.763,157.416
C02476=1057.163,390.883,-117.539,174.497,38.769,157.417
C02477=1057.171,391.129,-117.581,174.504,38.776,157.419
C02478=1057.179,391.376,-117.622,174.509,38.784,157.421
C02479=1057.187,391.622,-117.664,174.516,38.791,157.423
C02480=1057.194,391.868,-117.705,174.522,38.798,157.425
C02481=1057.203,392.115,-117.748,174.529,38.805,157.427
C02482=1057.211,392.361,-117.788,174.534,38.812,157.429
C02483=1057.219,392.607,-117.831,174.541,38.819,157.431
C02484=1057.226,392.853,-117.873,174.548,38.826,157.433
C02485=1057.234,393.099,-117.915,174.553,38.833,157.435
C02486=1057.242,393.346,-117.957,174.560,38.841,157.437
C02487=1057.251,393.592,-117.998,174.566,38.848,157.439
C02488=1057.259,393.838,-118.041,174.573,38.855,157.440
C02489=1057.266,394.084,-118.083,174.578,38.863,157.442
C02490=1057.275,394.331,-118.125,174.585,38.870,157.445
C02491=1057.282,394.577,-118.167,174.592,38.877,157.446
C02492=1057.290,394.824,-118.209,174.598,38.884,157.448
C02493=1057.298,395.069,-118.252,174.605,38.892,157.450
C02494=1057.306,395.316,-118.294,174.610,38.899,157.452
C02495=1057.314,395.562,-118.336,174.617,38.907,157.454
C02496=1057.323,395.808,-118.378,174.624,38.914,157.456
C02497=1057.331,396.053,-118.420,174.630,38.921,157.458
C02498=1057.339,396.300,-118.463,174.637,38.928,157.460
C02499=1057.347,396.547,-118.505,174.643,38.936,157.462
C02500=1057.355,396.793,-118.547,174.649,38.943,157.464
C02501=1057.363,397.039,-118.590,174.656,38.951,157.466
C02502=1057.372,397.286,-118.632,174.663,38.959,157.469
C02503=1057.379,397.531,-118.675,174.669,38.966,157.471
C02504=1057.388,397.778,-118.717,174.676,38.973,157.473
C02505=1057.396,398.024,-118.760,174.683,38.981,157.475
C02506=1057.403,398.270,-118.803,174.689,38.989,157.477
C02507=1057.412,398.516,-118.846,174.695,38.996,157.479
C02508=1057.420,398.762,-118.889,174.702,39.004,157.481
C02509=1057.428,399.009,-118.931,174.709,39.011,157.483
C02510=1057.436,399.254,-118.974,174.715,39.019,157.485
C02511=1057.445,399.500,-119.017,174.722,39.027,157.487
C02512=1057.453,399.747,-119.059,174.729,39.035,157.489
C02513=1057.461,399.993,-119.103,174.736,39.042,157.491
C02514=1057.469,400.239,-119.146,174.742,39.050,157.493
C02515=1057.478,400.485,-119.189,174.749,39.058,157.496
C02516=1057.485,400.731,-119.232,174.756,39.065,157.498
C02517=1057.494,400.977,-119.274,174.763,39.073,157.500
C02518=1057.502,401.223,-119.317,174.770,39.081,157.502
C02519=1057.510,401.470,-119.360,174.776,39.089,157.504
C02520=1057.524,401.848,-119.427,174.787,39.101,157.508
C02521=1057.536,402.227,-119.493,174.797,39.113,157.511
C02522=1057.549,402.606,-119.560,174.808,39.125,157.514
C02523=1057.562,402.984,-119.626,174.818,39.138,157.518
C02524=1057.569,403.230,-119.670,174.825,39.146,157.520
C02525=1057.578,403.477,-119.713,174.832,39.154,157.522
C02526=1057.587,403.722,-119.757,174.840,39.162,157.524
C02527=1057.595,403.969,-119.801,174.847,39.170,157.526
C02528=1057.603,404.215,-119.844,174.854,39.178,157.529
C02529=1057.612,404.460,-119.888,174.861,39.186,157.531
C02530=1057.620,404.706,-119.931,174.868,39.194,157.533
C02531=1057.629,404.952,-119.975,174.875,39.202,157.535
C02532=1057.637,405.198,-120.018,174.882,39.210,157.538
C02533=1057.645,405.444,-120.061,174.889,39.219,157.540
C02534=1057.654,405.691,-120.106,174.896,39.227,157.542
C02535=1057.662,405.937,-120.150,174.904,39.235,157.545
C02536=1057.670,406.183,-120.194,174.911,39.243,157.547
C02537=1057.678,406.428,-120.238,174.918,39.252,157.549
C02538=1057.687,406.674,-120.282,174.925,39.260,157.552
C02539=1057.696,406.921,-120.326,174.933,39.269,157.554
C02540=1057.703,407.144,-120.366,174.938,39.276,157.556
C02541=1057.711,407.367,-120.405,174.946,39.284,157.558
C02542=1057.718,407.590,-120.446,174.952,39.291,157.560
C02543=1057.726,407.815,-120.486,174.959,39.299,157.562
C02544=1057.733,408.038,-120.526,174.966,39.307,157.565
C02545=1057.742,408.261,-120.566,174.972,39.314,157.567
C02546=1057.749,408.485,-120.606,174.979,39.322,157.569
C02547=1057.757,408.708,-120.646,174.986,39.330,157.571
C02548=1057.766,408.954,-120.691,174.993,39.338,157.573
C02549=1057.774,409.200,-120.735,175.000,39.346,157.576
C02550=1057.783,409.446,-120.780,175.008,39.355,157.578
C02551=1057.792,409.691,-120.823,175.015,39.364,157.581
C02552=1057.800,409.937,-120.868,175.023,39.373,157.583
C02553=1057.809,410.183,-120.913,175.031,39.381,157.585
C02554=1057.817,410.428,-120.957,175.038,39.390,157.588
C02555=1057.826,410.675,-121.002,175.045,39.399,157.590
C02556=1057.834,410.921,-121.046,175.053,39.407,157.593
C02557=1057.844,411.166,-121.091,175.061,39.416,157.595
C02558=1057.853,411.413,-121.135,175.068,39.425,157.598
C02559=1057.861,411.658,-121.180,175.076,39.434,157.600
C02560=1057.870,411.904,-121.225,175.083,39.442,157.603
C02561=1057.878,412.150,-121.269,175.092,39.451,157.605
C02562=1057.887,412.395,-121.314,175.099,39.459,157.608
C02563=1057.896,412.642,-121.359,175.106,39.468,157.610
C02564=1057.905,412.887,-121.403,175.115,39.478,157.613
C02565=1057.914,413.133,-121.448,175.122,39.486,157.615
C02566=1057.923,413.379,-121.494,175.130,39.495,157.618
C02567=1057.931,413.625,-121.538,175.138,39.504,157.620
C02568=1057.940,413.871,-121.583,175.146,39.513,157.623
C02569=1057.949,414.116,-121.629,175.154,39.522,157.626
C02570=1057.958,414.362,-121.674,175.162,39.531,157.628
C02571=1057.966,414.609,-121.719,175.169,39.540,157.631
C02572=1057.975,414.854,-121.764,175.178,39.550,157.633
C02573=1057.984,415.100,-121.809,175.185,39.558,157.636
C02574=1057.993,415.345,-121.855,175.194,39.568,157.639
C02575=1058.002,415.591,-121.900,175.202,39.577,157.641
C02576=1058.014,415.930,-121.963,175.213,39.589,157.645
C02577=1058.026,416.269,-122.026,175.224,39.602,157.649
C02578=1058.039,416.608,-122.089,175.235,39.615,157.652
C02579=1058.051,416.947,-122.151,175.247,39.628,157.656
C02580=1058.060,417.193,-122.197,175.255,39.638,157.659
C02581=1058.068,417.439,-122.243,175.263,39.647,157.661
C02582=1058.077,417.685,-122.288,175.271,39.656,157.664
C02583=1058.087,417.930,-122.334,175.280,39.666,157.667
C02584=1058.096,418.176,-122.380,175.288,39.675,157.670
C02585=1058.105,418.421,-122.426,175.296,39.684,157.672
C02586=1058.114,418.667,-122.471,175.305,39.694,157.675
C02587=1058.123,418.912,-122.517,175.313,39.703,157.678
C02588=1058.132,419.158,-122.563,175.322,39.713,157.681
C02589=1058.142,419.403,-122.609,175.330,39.723,157.683
C02590=1058.151,419.649,-122.654,175.338,39.732,157.686
C02591=1058.160,419.895,-122.702,175.347,39.742,157.689
C02592=1058.169,420.141,-122.748,175.356,39.752,157.692
C02593=1058.178,420.387,-122.793,175.365,39.761,157.695
C02594=1058.186,420.632,-122.840,175.372,39.771,157.697
C02595=1058.196,420.877,-122.886,175.381,39.781,157.700
C02596=1058.205,421.122,-122.932,175.390,39.791,157.703
C02597=1058.214,421.369,-122.979,175.399,39.800,157.706
C02598=1058.223,421.614,-123.025,175.407,39.810,157.709
C02599=1058.233,421.859,-123.071,175.416,39.820,157.712
C02600=1058.241,422.105,-123.118,175.425,39.830,157.715
C02601=1058.251,422.350,-123.165,175.434,39.840,157.718
C02602=1058.260,422.596,-123.211,175.443,39.850,157.721
C02603=1058.269,422.841,-123.258,175.452,39.860,157.724
C02604=1058.279,423.086,-123.305,175.461,39.870,157.726
C02605=1058.288,423.332,-123.351,175.469,39.880,157.729
C02606=1058.297,423.577,-123.398,175.478,39.891,157.732
C02607=1058.306,423.823,-123.445,175.487,39.900,157.735
C02608=1058.316,424.068,-123.492,175.496,39.910,157.738
C02609=1058.326,424.314,-123.538,175.505,39.921,157.741
C02610=1058.334,424.559,-123.586,175.514,39.931,157.744
C02611=1058.344,424.805,-123.632,175.523,39.941,157.747
C02612=1058.353,425.050,-123.679,175.532,39.951,157.750
C02613=1058.363,425.295,-123.726,175.541,39.962,157.754
C02614=1058.372,425.540,-123.773,175.550,39.972,157.757
C02615=1058.382,425.786,-123.820,175.559,39.982,157.760
C02616=1058.391,426.032,-123.868,175.569,39.992,157.763
C02617=1058.401,426.276,-123.915,175.579,40.003,157.766
C02618=1058.410,426.522,-123.962,175.588,40.013,157.769
C02619=1058.420,426.767,-124.009,175.597,40.024,157.772
C02620=1058.429,427.013,-124.056,175.606,40.035,157.775
C02621=1058.439,427.258,-124.104,175.616,40.045,157.778
C02622=1058.448,427.503,-124.151,175.625,40.055,157.781
C02623=1058.458,427.749,-124.199,175.635,40.066,157.785
C02624=1058.467,427.994,-124.247,175.644,40.077,157.788
C02625=1058.477,428.239,-124.295,175.654,40.087,157.791
C02626=1058.486,428.484,-124.342,175.663,40.099,157.794
C02627=1058.496,428.729,-124.390,175.673,40.109,157.798
C02628=1058.505,428.975,-124.438,175.683,40.120,157.801
C02629=1058.516,429.220,-124.486,175.692,40.130,157.804
C02630=1058.525,429.465,-124.533,175.702,40.142,157.807
C02631=1058.534,429.710,-124.581,175.712,40.152,157.811
C02632=1058.549,430.070,-124.651,175.726,40.168,157.815
C02633=1058.563,430.431,-124.722,175.740,40.184,157.820
C02634=1058.577,430.791,-124.793,175.755,40.201,157.825
C02635=1058.592,431.151,-124.864,175.769,40.217,157.830
C02636=1058.601,431.397,-124.912,175.780,40.228,157.833
C02637=1058.611,431.642,-124.960,175.789,40.239,157.837
C02638=1058.621,431.887,-125.009,175.800,40.250,157.840
C02639=1058.630,432.132,-125.057,175.810,40.262,157.844
C02640=1058.640,432.377,-125.106,175.820,40.273,157.847
C02641=1058.650,432.622,-125.154,175.830,40.284,157.851
C02642=1058.660,432.867,-125.203,175.840,40.295,157.854
C02643=1058.670,433.112,-125.252,175.850,40.307,157.857
C02644=1058.680,433.357,-125.300,175.861,40.318,157.861
C02645=1058.689,433.602,-125.349,175.871,40.329,157.864
C02646=1058.699,433.847,-125.397,175.881,40.341,157.868
C02647=1058.709,434.092,-125.447,175.892,40.352,157.871
C02648=1058.720,434.337,-125.496,175.902,40.364,157.875
C02649=1058.729,434.582,-125.544,175.912,40.375,157.879
C02650=1058.739,434.827,-125.593,175.923,40.387,157.882
C02651=1058.749,435.072,-125.642,175.934,40.398,157.886
C02652=1058.760,435.317,-125.691,175.944,40.410,157.889
C02653=1058.770,435.562,-125.740,175.955,40.422,157.893
C02654=1058.780,435.807,-125.790,175.966,40.433,157.896
C02655=1058.790,436.052,-125.838,175.976,40.445,157.900
C02656=1058.800,436.296,-125.887,175.987,40.457,157.904
C02657=1058.811,436.541,-125.937,175.997,40.469,157.907
C02658=1058.821,436.786,-125.986,176.008,40.481,157.911
C02659=1058.831,437.031,-126.035,176.019,40.493,157.915
C02660=1058.841,437.275,-126.084,176.030,40.504,157.918
C02661=1058.852,437.520,-126.134,176.041,40.517,157.922
C02662=1058.862,437.766,-126.184,176.052,40.529,157.926
C02663=1058.872,438.010,-126.233,176.063,40.541,157.930
C02664=1058.883,438.255,-126.283,176.074,40.552,157.934
C02665=1058.893,438.500,-126.332,176.086,40.565,157.937
C02666=1058.903,438.745,-126.382,176.097,40.577,157.941
C02667=1058.914,438.989,-126.433,176.108,40.589,157.945
C02668=1058.924,439.234,-126.482,176.119,40.601,157.949
C02669=1058.934,439.479,-126.532,176.130,40.614,157.953
C02670=1058.945,439.723,-126.583,176.141,40.626,157.957
C02671=1058.955,439.969,-126.632,176.154,40.638,157.961
C02672=1058.965,440.213,-126.683,176.165,40.651,157.964
C02673=1058.976,440.458,-126.732,176.176,40.663,157.968
C02674=1058.986,440.702,-126.783,176.187,40.676,157.972
C02675=1058.997,440.947,-126.834,176.199,40.688,157.976
C02676=1059.007,441.192,-126.883,176.211,40.700,157.980
C02677=1059.017,441.436,-126.934,176.223,40.713,157.984
C02678=1059.028,441.680,-126.984,176.234,40.726,157.988
C02679=1059.038,441.925,-127.035,176.245,40.739,157.992
C02680=1059.049,442.169,-127.085,176.258,40.751,157.996
C02681=1059.059,442.414,-127.136,176.269,40.764,158.000
C02682=1059.070,442.659,-127.187,176.282,40.777,158.005
C02683=1059.081,442.903,-127.237,176.293,40.790,158.009
C02684=1059.092,443.148,-127.288,176.305,40.803,158.013
C02685=1059.102,443.393,-127.339,176.317,40.816,158.017
C02686=1059.114,443.637,-127.390,176.329,40.829,158.021
C02687=1059.124,443.882,-127.441,176.342,40.841,158.025
C02688=1059.137,444.188,-127.505,176.356,40.858,158.030
C02689=1059.151,444.494,-127.568,176.372,40.874,158.036
C02690=1059.164,444.800,-127.632,176.387,40.891,158.041
C02691=1059.178,445.107,-127.697,176.403,40.907,158.046
C02692=1059.189,445.351,-127.748,176.415,40.921,158.051
C02693=1059.200,445.596,-127.799,176.428,40.934,158.055
C02694=1059.211,445.840,-127.851,176.440,40.947,158.059
C02695=1059.222,446.084,-127.902,176.453,40.961,158.064
C02696=1059.233,446.329,-127.954,176.465,40.974,158.068
C02697=1059.244,446.573,-128.005,176.478,40.988,158.072
C02698=1059.255,446.817,-128.057,176.491,41.001,158.077
C02699=1059.266,447.062,-128.109,176.504,41.014,158.081
C02700=1059.278,447.304,-128.159,176.517,41.028,158.086
C02701=1059.290,447.547,-128.210,176.530,41.041,158.090
C02702=1059.304,447.791,-128.259,176.543,41.054,158.094
C02703=1059.318,448.036,-128.309,176.555,41.067,158.098
C02704=1059.333,448.280,-128.357,176.569,41.079,158.103
C02705=1059.349,448.524,-128.405,176.582,41.092,158.107
C02706=1059.367,448.769,-128.453,176.595,41.103,158.111
C02707=1059.384,449.014,-128.500,176.609,41.115,158.115
C02708=1059.403,449.259,-128.546,176.622,41.126,158.119
C02709=1059.422,449.504,-128.591,176.635,41.138,158.122
C02710=1059.443,449.750,-128.636,176.650,41.149,158.126
C02711=1059.464,449.994,-128.681,176.663,41.160,158.130
C02712=1059.134,450.008,-128.962,176.659,41.271,158.161
C02713=1059.113,449.763,-128.917,176.645,41.260,158.157
C02714=1059.093,449.517,-128.872,176.631,41.249,158.153
C02715=1059.073,449.272,-128.827,176.617,41.238,158.149
C02716=1059.054,449.027,-128.780,176.603,41.226,158.145
C02717=1059.036,448.782,-128.734,176.590,41.215,158.141
C02718=1059.019,448.537,-128.686,176.577,41.203,158.137
C02719=1059.003,448.293,-128.638,176.564,41.191,158.133
C02720=1058.987,448.049,-128.590,176.550,41.178,158.129
C02721=1058.973,447.804,-128.540,176.537,41.166,158.125
C02722=1058.960,447.560,-128.490,176.524,41.153,158.121
C02723=1058.947,447.317,-128.440,176.511,41.140,158.116
C02724=1058.934,447.074,-128.389,176.498,41.127,158.112
C02725=1058.924,446.830,-128.338,176.485,41.113,158.108
C02726=1058.912,446.585,-128.286,176.472,41.100,158.103
C02727=1058.901,446.341,-128.234,176.459,41.086,158.099
C02728=1058.890,446.097,-128.183,176.447,41.073,158.094
C02729=1058.880,445.853,-128.132,176.435,41.060,158.090
C02730=1058.868,445.609,-128.080,176.422,41.046,158.086
C02731=1058.857,445.365,-128.029,176.409,41.033,158.081
C02732=1058.847,445.120,-127.978,176.396,41.020,158.077
C02733=1058.834,444.832,-127.917,176.381,41.005,158.072
C02734=1058.821,444.545,-127.857,176.367,40.989,158.067
C02735=1058.807,444.259,-127.797,176.352,40.974,158.062
C02736=1058.795,443.972,-127.737,176.339,40.958,158.057
C02737=1058.784,443.727,-127.686,176.326,40.946,158.053
C02738=1058.774,443.482,-127.635,176.314,40.932,158.049
C02739=1058.763,443.238,-127.584,176.302,40.920,158.045
C02740=1058.753,442.994,-127.533,176.290,40.907,158.041
C02741=1058.742,442.749,-127.483,176.277,40.894,158.036
C02742=1058.731,442.504,-127.432,176.266,40.881,158.032
C02743=1058.720,442.260,-127.382,176.253,40.869,158.028
C02744=1058.710,442.015,-127.331,176.242,40.856,158.024
C02745=1058.699,441.771,-127.280,176.230,40.843,158.020
C02746=1058.688,441.526,-127.230,176.218,40.831,158.016
C02747=1058.678,441.282,-127.179,176.206,40.818,158.012
C02748=1058.667,441.037,-127.129,176.195,40.806,158.008
C02749=1058.657,440.792,-127.078,176.183,40.793,158.004
C02750=1058.646,440.547,-127.028,176.171,40.781,158.000
C02751=1058.635,440.303,-126.978,176.160,40.768,157.996
C02752=1058.625,440.059,-126.927,176.149,40.756,157.992
C02753=1058.615,439.814,-126.878,176.137,40.743,157.988
C02754=1058.605,439.569,-126.827,176.125,40.731,157.984
C02755=1058.594,439.324,-126.777,176.114,40.719,157.980
C02756=1058.584,439.080,-126.728,176.103,40.707,157.977
C02757=1058.573,438.835,-126.678,176.091,40.694,157.973
C02758=1058.563,438.590,-126.628,176.080,40.683,157.969
C02759=1058.553,438.346,-126.578,176.069,40.670,157.965
C02760=1058.542,438.101,-126.529,176.058,40.658,157.961
C02761=1058.531,437.855,-126.479,176.047,40.646,157.958
C02762=1058.522,437.611,-126.429,176.036,40.634,157.954
C02763=1058.511,437.366,-126.379,176.025,40.622,157.950
C02764=1058.501,437.121,-126.330,176.014,40.611,157.946
C02765=1058.491,436.876,-126.281,176.003,40.599,157.943
C02766=1058.480,436.631,-126.231,175.991,40.587,157.939
C02767=1058.470,436.387,-126.182,175.980,40.575,157.935
C02768=1058.459,436.142,-126.132,175.970,40.563,157.932
C02769=1058.450,435.897,-126.084,175.960,40.551,157.928
C02770=1058.440,435.653,-126.035,175.949,40.540,157.924
C02771=1058.429,435.408,-125.985,175.938,40.528,157.921
C02772=1058.419,435.163,-125.936,175.927,40.516,157.917
C02773=1058.408,434.918,-125.887,175.916,40.505,157.913
C02774=1058.399,434.673,-125.838,175.906,40.493,157.910
C02775=1058.389,434.428,-125.789,175.895,40.482,157.906
C02776=1058.378,434.183,-125.740,175.885,40.470,157.903
C02777=1058.368,433.938,-125.692,175.875,40.459,157.899
C02778=1058.359,433.693,-125.643,175.864,40.448,157.896
C02779=1058.349,433.448,-125.594,175.853,40.436,157.892
C02780=1058.339,433.203,-125.545,175.843,40.425,157.889
C02781=1058.329,432.958,-125.496,175.833,40.414,157.885
C02782=1058.319,432.713,-125.448,175.822,40.402,157.882
C02783=1058.309,432.468,-125.399,175.812,40.391,157.878
C02784=1058.299,432.223,-125.351,175.802,40.380,157.875
C02785=1058.290,431.978,-125.302,175.792,40.369,157.871
C02786=1058.280,431.733,-125.254,175.781,40.358,157.868
C02787=1058.270,431.488,-125.205,175.772,40.347,157.865
C02788=1058.260,431.243,-125.157,175.761,40.336,157.861
C02789=1058.246,430.880,-125.085,175.747,40.319,157.856
C02790=1058.232,430.518,-125.014,175.732,40.303,157.851
C02791=1058.217,430.155,-124.943,175.718,40.287,157.846
C02792=1058.203,429.793,-124.871,175.702,40.271,157.841
C02793=1058.193,429.547,-124.824,175.693,40.260,157.838
C02794=1058.183,429.302,-124.776,175.683,40.249,157.835
C02795=1058.174,429.058,-124.728,175.673,40.238,157.832
C02796=1058.164,428.812,-124.680,175.664,40.228,157.828
C02797=1058.154,428.567,-124.633,175.654,40.217,157.825
C02798=1058.145,428.322,-124.585,175.645,40.206,157.822
C02799=1058.135,428.076,-124.537,175.635,40.196,157.819
C02800=1058.125,427.832,-124.490,175.625,40.185,157.816
C02801=1058.116,427.586,-124.442,175.616,40.174,157.812
C02802=1058.107,427.341,-124.394,175.607,40.164,157.809
C02803=1058.096,427.095,-124.347,175.596,40.153,157.806
C02804=1058.088,426.850,-124.300,175.587,40.143,157.803
C02805=1058.078,426.605,-124.252,175.578,40.132,157.800
C02806=1058.068,426.360,-124.205,175.568,40.122,157.797
C02807=1058.059,426.115,-124.157,175.559,40.112,157.793
C02808=1058.049,425.869,-124.111,175.550,40.101,157.790
C02809=1058.040,425.624,-124.063,175.541,40.091,157.787
C02810=1058.030,425.379,-124.016,175.532,40.081,157.784
C02811=1058.021,425.133,-123.968,175.522,40.070,157.781
C02812=1058.011,424.888,-123.922,175.512,40.060,157.778
C02813=1058.002,424.642,-123.874,175.503,40.050,157.775
C02814=1057.993,424.397,-123.828,175.494,40.040,157.772
C02815=1057.983,424.151,-123.780,175.485,40.030,157.769
C02816=1057.974,423.906,-123.734,175.476,40.020,157.766
C02817=1057.964,423.660,-123.688,175.467,40.009,157.763
C02818=1057.955,423.415,-123.640,175.459,40.000,157.760
C02819=1057.945,423.169,-123.594,175.450,39.989,157.757
C02820=1057.937,422.924,-123.547,175.441,39.979,157.754
C02821=1057.927,422.679,-123.500,175.432,39.969,157.751
C02822=1057.917,422.433,-123.454,175.423,39.959,157.748
C02823=1057.909,422.188,-123.407,175.414,39.950,157.745
C02824=1057.899,421.943,-123.361,175.405,39.940,157.742
C02825=1057.890,421.697,-123.314,175.396,39.930,157.739
C02826=1057.881,421.451,-123.268,175.387,39.920,157.737
C02827=1057.872,421.206,-123.222,175.379,39.910,157.734
C02828=1057.863,420.961,-123.175,175.370,39.900,157.731
C02829=1057.853,420.715,-123.128,175.361,39.891,157.728
C02830=1057.844,420.469,-123.082,175.352,39.881,157.725
C02831=1057.835,420.224,-123.035,175.344,39.871,157.722
C02832=1057.826,419.979,-122.989,175.335,39.861,157.719
C02833=1057.817,419.733,-122.944,175.327,39.852,157.717
C02834=1057.808,419.488,-122.898,175.318,39.843,157.714
C02835=1057.798,419.242,-122.851,175.310,39.833,157.711
C02836=1057.790,418.996,-122.805,175.301,39.823,157.708
C02837=1057.781,418.750,-122.759,175.292,39.814,157.705
C02838=1057.772,418.505,-122.714,175.285,39.804,157.703
C02839=1057.762,418.259,-122.668,175.276,39.795,157.700
C02840=1057.753,418.014,-122.622,175.267,39.786,157.697
C02841=1057.744,417.768,-122.576,175.259,39.776,157.694
C02842=1057.735,417.523,-122.531,175.251,39.766,157.692
C02843=1057.726,417.277,-122.485,175.243,39.757,157.689
C02844=1057.717,417.031,-122.440,175.234,39.748,157.686
C02845=1057.704,416.690,-122.376,175.222,39.735,157.683
C02846=1057.692,416.349,-122.312,175.212,39.722,157.679
C02847=1057.680,416.008,-122.249,175.200,39.709,157.675
C02848=1057.668,415.666,-122.186,175.188,39.697,157.671
C02849=1057.659,415.420,-122.141,175.181,39.688,157.669
C02850=1057.650,415.175,-122.096,175.172,39.678,157.666
C02851=1057.641,414.929,-122.051,175.164,39.669,157.663
C02852=1057.632,414.684,-122.005,175.157,39.660,157.661
C02853=1057.623,414.438,-121.960,175.148,39.651,157.658
C02854=1057.614,414.192,-121.914,175.141,39.642,157.656
C02855=1057.606,413.947,-121.869,175.132,39.633,157.653
C02856=1057.597,413.701,-121.824,175.125,39.624,157.650
C02857=1057.588,413.454,-121.779,175.116,39.615,157.648
C02858=1057.579,413.209,-121.734,175.109,39.606,157.645
C02859=1057.570,412.964,-121.689,175.101,39.598,157.643
C02860=1057.561,412.717,-121.645,175.093,39.588,157.640
C02861=1057.552,412.472,-121.599,175.085,39.579,157.638
C02862=1057.544,412.226,-121.555,175.078,39.571,157.635
C02863=1057.535,411.980,-121.510,175.069,39.562,157.633
C02864=1057.526,411.734,-121.465,175.062,39.553,157.630
C02865=1057.518,411.489,-121.420,175.054,39.545,157.628
C02866=1057.508,411.243,-121.376,175.047,39.536,157.625
C02867=1057.500,410.997,-121.332,175.039,39.527,157.623
C02868=1057.491,410.751,-121.286,175.031,39.519,157.620
C02869=1057.482,410.505,-121.242,175.024,39.510,157.618
C02870=1057.474,410.259,-121.198,175.016,39.501,157.616
C02871=1057.465,410.013,-121.153,175.008,39.493,157.613
C02872=1057.456,409.768,-121.109,175.001,39.484,157.611
C02873=1057.447,409.521,-121.064,174.993,39.475,157.608
C02874=1057.439,409.276,-121.020,174.986,39.467,157.606
C02875=1057.430,409.030,-120.976,174.979,39.458,157.603
C02876=1057.422,408.784,-120.931,174.970,39.450,157.601
C02877=1057.414,408.538,-120.887,174.963,39.442,157.599
C02878=1057.404,408.292,-120.843,174.956,39.433,157.596
C02879=1057.396,408.046,-120.798,174.948,39.425,157.594
C02880=1057.388,407.800,-120.754,174.941,39.416,157.591
C02881=1057.379,407.554,-120.710,174.934,39.408,157.589
C02882=1057.371,407.309,-120.666,174.927,39.399,157.587
C02883=1057.363,407.062,-120.622,174.919,39.391,157.584
C02884=1057.353,406.816,-120.578,174.912,39.383,157.582
C02885=1057.345,406.570,-120.534,174.905,39.375,157.580
C02886=1057.337,406.325,-120.490,174.898,39.366,157.577
C02887=1057.329,406.079,-120.446,174.890,39.358,157.575
C02888=1057.321,405.833,-120.402,174.883,39.350,157.573
C02889=1057.311,405.587,-120.358,174.876,39.341,157.570
C02890=1057.304,405.340,-120.314,174.869,39.333,157.568
C02891=1057.295,405.095,-120.270,174.862,39.325,157.566
C02892=1057.287,404.848,-120.227,174.855,39.317,157.564
C02893=1057.278,404.603,-120.183,174.847,39.309,157.561
C02894=1057.270,404.356,-120.139,174.840,39.301,157.559
C02895=1057.261,404.110,-120.096,174.833,39.293,157.557
C02896=1057.253,403.865,-120.052,174.826,39.285,157.555
C02897=1057.245,403.618,-120.009,174.819,39.277,157.552
C02898=1057.236,403.372,-119.966,174.812,39.269,157.550
C02899=1057.228,403.126,-119.921,174.805,39.261,157.548
C02900=1057.220,402.880,-119.878,174.797,39.253,157.546
C02901=1057.208,402.545,-119.820,174.788,39.242,157.543
C02902=1057.197,402.209,-119.761,174.779,39.231,157.540
C02903=1057.186,401.873,-119.702,174.769,39.221,157.537
C02904=1057.174,401.539,-119.642,174.760,39.209,157.534
C02905=1057.165,401.293,-119.599,174.753,39.202,157.532
C02906=1057.157,401.046,-119.556,174.746,39.194,157.529
C02907=1057.149,400.799,-119.513,174.739,39.186,157.527
C02908=1057.141,400.553,-119.470,174.732,39.178,157.525
C02909=1057.132,400.307,-119.427,174.725,39.171,157.523
C02910=1057.124,400.062,-119.385,174.719,39.163,157.521
C02911=1057.116,399.816,-119.342,174.712,39.156,157.519
C02912=1057.108,399.570,-119.298,174.705,39.148,157.517
C02913=1057.100,399.323,-119.256,174.698,39.140,157.515
C02914=1057.091,399.077,-119.213,174.692,39.133,157.513
C02915=1057.083,398.831,-119.170,174.685,39.125,157.510
C02916=1057.075,398.585,-119.128,174.678,39.117,157.508
C02917=1057.067,398.339,-119.085,174.671,39.110,157.506
C02918=1057.058,398.093,-119.042,174.665,39.102,157.504
C02919=1057.051,397.847,-119.000,174.659,39.095,157.502
C02920=1057.043,397.600,-118.956,174.652,39.087,157.500
C02921=1057.035,397.354,-118.914,174.646,39.080,157.498
C02922=1057.026,397.108,-118.871,174.639,39.072,157.496
C02923=1057.019,396.862,-118.829,174.632,39.064,157.494
C02924=1057.010,396.616,-118.786,174.626,39.057,157.492
C02925=1057.003,396.404,-118.750,174.620,39.051,157.490
C02926=1056.996,396.193,-118.713,174.614,39.044,157.488
C02927=1056.989,395.981,-118.678,174.608,39.038,157.487
C02928=1056.982,395.770,-118.640,174.604,39.032,157.485
C02929=1056.975,395.558,-118.604,174.598,39.026,157.483
C02930=1056.968,395.347,-118.568,174.593,39.019,157.482
C02931=1056.961,395.136,-118.532,174.587,39.013,157.480
C02932=1056.954,394.925,-118.496,174.581,39.007,157.478
C02933=1056.946,394.679,-118.453,174.575,38.999,157.476
C02934=1056.938,394.432,-118.411,174.568,38.992,157.474
C02935=1056.930,394.186,-118.369,174.562,38.985,157.472
C02936=1056.922,393.939,-118.327,174.555,38.978,157.470
C02937=1056.915,393.693,-118.285,174.549,38.971,157.468
C02938=1056.907,393.447,-118.243,174.543,38.963,157.466
C02939=1056.898,393.201,-118.201,174.536,38.956,157.464
C02940=1056.890,392.955,-118.159,174.530,38.949,157.462
C02941=1056.882,392.708,-118.117,174.523,38.942,157.461
C02942=1056.875,392.462,-118.075,174.518,38.935,157.459
C02943=1056.866,392.216,-118.033,174.511,38.928,157.457
C02944=1056.858,391.970,-117.991,174.505,38.921,157.455
C02945=1056.851,391.723,-117.950,174.498,38.913,157.453
C02946=1056.843,391.477,-117.908,174.493,38.906,157.451
C02947=1056.834,391.231,-117.867,174.486,38.899,157.449
C02948=1056.827,390.985,-117.825,174.480,38.893,157.447
C02949=1056.819,390.738,-117.783,174.473,38.885,157.445
C02950=1056.811,390.492,-117.741,174.468,38.878,157.443
C02951=1056.803,390.246,-117.700,174.461,38.871,157.441
C02952=1056.795,389.999,-117.658,174.455,38.864,157.440
C02953=1056.787,389.753,-117.616,174.449,38.857,157.438
C02954=1056.779,389.507,-117.576,174.443,38.850,157.436
C02955=1056.771,389.260,-117.533,174.436,38.844,157.434
C02956=1056.763,389.014,-117.493,174.431,38.837,157.432
C02957=1056.751,388.626,-117.428,174.421,38.826,157.429
C02958=1056.738,388.239,-117.363,174.412,38.815,157.426
C02959=1056.725,387.852,-117.298,174.402,38.805,157.424
C02960=1056.713,387.464,-117.233,174.393,38.794,157.421
C02961=1056.705,387.217,-117.192,174.387,38.787,157.419
C02962=1056.697,386.971,-117.150,174.380,38.781,157.417
C02963=1056.689,386.724,-117.110,174.375,38.774,157.415
C02964=1056.681,386.478,-117.069,174.369,38.767,157.414
C02965=1056.674,386.231,-117.028,174.363,38.761,157.412
C02966=1056.666,385.986,-116.987,174.357,38.754,157.410
C02967=1056.658,385.739,-116.945,174.351,38.747,157.408
C02968=1056.650,385.493,-116.905,174.345,38.741,157.407
C02969=1056.642,385.246,-116.863,174.339,38.734,157.405
C02970=1056.634,384.999,-116.823,174.334,38.728,157.403
C02971=1056.626,384.753,-116.782,174.327,38.721,157.401
C02972=1056.619,384.506,-116.741,174.322,38.714,157.399
C02973=1056.611,384.260,-116.700,174.316,38.708,157.398
C02974=1056.603,384.013,-116.660,174.310,38.701,157.396
C02975=1056.596,383.767,-116.619,174.304,38.695,157.394
C02976=1056.588,383.520,-116.578,174.298,38.688,157.393
C02977=1056.581,383.274,-116.537,174.293,38.681,157.391
C02978=1056.573,383.028,-116.497,174.286,38.675,157.389
C02979=1056.565,382.782,-116.456,174.281,38.669,157.387
C02980=1056.558,382.535,-116.416,174.275,38.662,157.386
C02981=1056.550,382.288,-116.375,174.270,38.656,157.384
C02982=1056.542,382.042,-116.334,174.264,38.649,157.382
C02983=1056.535,381.795,-116.294,174.258,38.643,157.381
C02984=1056.527,381.549,-116.253,174.253,38.636,157.379
C02985=1056.519,381.302,-116.213,174.247,38.630,157.377
C02986=1056.512,381.055,-116.172,174.242,38.623,157.376
C02987=1056.505,380.810,-116.132,174.236,38.617,157.374
C02988=1056.497,380.563,-116.092,174.230,38.611,157.372
C02989=1056.490,380.316,-116.051,174.224,38.605,157.371
C02990=1056.482,380.069,-116.011,174.219,38.598,157.369
C02991=1056.474,379.823,-115.970,174.213,38.592,157.367
C02992=1056.466,379.576,-115.930,174.208,38.586,157.366
C02993=1056.459,379.330,-115.891,174.201,38.579,157.364
C02994=1056.452,379.083,-115.851,174.196,38.573,157.362
C02995=1056.444,378.837,-115.810,174.191,38.567,157.361
C02996=1056.436,378.590,-115.770,174.185,38.561,157.359
C02997=1056.428,378.343,-115.730,174.180,38.554,157.357
C02998=1056.421,378.096,-115.691,174.175,38.548,157.356
C02999=1056.413,377.850,-115.650,174.169,38.542,157.354
C03000=1056.405,377.603,-115.610,174.163,38.536,157.353
C03001=1056.398,377.356,-115.570,174.157,38.530,157.351
C03002=1056.390,377.110,-115.531,174.152,38.524,157.349
C03003=1056.383,376.863,-115.491,174.147,38.518,157.348
C03004=1056.375,376.616,-115.451,174.141,38.512,157.346
C03005=1056.368,376.370,-115.411,174.136,38.506,157.345
C03006=1056.360,376.123,-115.371,174.130,38.499,157.343
C03007=1056.352,375.876,-115.331,174.125,38.493,157.342
C03008=1056.345,375.630,-115.292,174.120,38.487,157.340
C03009=1056.338,375.383,-115.252,174.114,38.481,157.338
C03010=1056.330,375.136,-115.212,174.109,38.476,157.337
C03011=1056.323,374.890,-115.172,174.104,38.469,157.335
C03012=1056.315,374.643,-115.133,174.098,38.463,157.334
C03013=1056.307,374.358,-115.087,174.092,38.456,157.332
C03014=1056.298,374.071,-115.040,174.085,38.450,157.330
C03015=1056.289,373.785,-114.995,174.080,38.442,157.328
C03016=1056.281,373.499,-114.950,174.073,38.435,157.327
C03017=1056.273,373.252,-114.910,174.068,38.430,157.325
C03018=1056.266,373.006,-114.870,174.063,38.424,157.323
C03019=1056.259,372.758,-114.831,174.057,38.418,157.322
C03020=1056.252,372.512,-114.792,174.052,38.412,157.320
C03021=1056.244,372.265,-114.752,174.047,38.406,157.319
C03022=1056.237,372.018,-114.713,174.042,38.400,157.317
C03023=1056.229,371.772,-114.673,174.036,38.394,157.316
C03024=1056.222,371.525,-114.635,174.031,38.388,157.314
C03025=1056.214,371.278,-114.595,174.026,38.383,157.313
C03026=1056.207,371.031,-114.556,174.020,38.377,157.311
C03027=1056.199,370.784,-114.517,174.015,38.371,157.310
C03028=1056.192,370.538,-114.478,174.010,38.365,157.308
C03029=1056.184,370.290,-114.439,174.005,38.360,157.307
C03030=1056.177,370.044,-114.400,174.000,38.354,157.306
C03031=1056.170,369.797,-114.361,173.995,38.348,157.304
C03032=1056.162,369.550,-114.322,173.990,38.343,157.303
C03033=1056.155,369.304,-114.283,173.985,38.337,157.301
C03034=1056.147,369.057,-114.244,173.980,38.331,157.300
C03035=1056.140,368.810,-114.205,173.974,38.325,157.298
C03036=1056.133,368.563,-114.166,173.969,38.320,157.297
C03037=1056.124,368.316,-114.127,173.964,38.314,157.295
C03038=1056.118,368.070,-114.088,173.959,38.308,157.294
C03039=1056.111,367.823,-114.049,173.954,38.303,157.292
C03040=1056.103,367.576,-114.011,173.948,38.297,157.291
C03041=1056.096,367.329,-113.972,173.944,38.291,157.289
C03042=1056.088,367.082,-113.934,173.939,38.286,157.288
C03043=1056.082,366.835,-113.895,173.934,38.280,157.287
C03044=1056.073,366.588,-113.856,173.929,38.275,157.285
C03045=1056.067,366.341,-113.817,173.923,38.269,157.284
C03046=1056.060,366.095,-113.778,173.918,38.264,157.282
C03047=1056.052,365.848,-113.740,173.914,38.258,157.281
C03048=1056.045,365.600,-113.701,173.909,38.252,157.279
C03049=1056.037,365.354,-113.663,173.904,38.247,157.278
C03050=1056.030,365.107,-113.624,173.898,38.241,157.277
C03051=1056.023,364.861,-113.586,173.893,38.236,157.275
C03052=1056.016,364.614,-113.547,173.889,38.230,157.274
C03053=1056.010,364.366,-113.509,173.884,38.225,157.273
C03054=1056.001,364.119,-113.470,173.879,38.219,157.271
C03055=1055.995,363.872,-113.431,173.874,38.214,157.270
C03056=1055.987,363.626,-113.393,173.869,38.208,157.268
C03057=1055.981,363.378,-113.355,173.864,38.203,157.267
C03058=1055.973,363.132,-113.317,173.859,38.198,157.266
C03059=1055.965,362.885,-113.278,173.854,38.192,157.264
C03060=1055.959,362.638,-113.240,173.849,38.187,157.263
C03061=1055.951,362.391,-113.202,173.845,38.181,157.261
C03062=1055.944,362.144,-113.164,173.840,38.176,157.260
C03063=1055.937,361.897,-113.125,173.835,38.171,157.259
C03064=1055.929,361.650,-113.087,173.830,38.165,157.257
C03065=1055.922,361.403,-113.050,173.826,38.160,157.256
C03066=1055.915,361.156,-113.012,173.820,38.155,157.255
C03067=1055.908,360.909,-112.973,173.815,38.149,157.253
C03068=1055.901,360.662,-112.936,173.810,38.144,157.252
C03069=1055.893,360.395,-112.895,173.805,38.138,157.251
C03070=1055.885,360.127,-112.854,173.800,38.132,157.249
C03071=1055.877,359.859,-112.812,173.795,38.127,157.248
C03072=1055.869,359.592,-112.771,173.790,38.121,157.246
C03073=1055.862,359.345,-112.733,173.786,38.116,157.245
C03074=1055.855,359.097,-112.696,173.780,38.110,157.244
C03075=1055.847,358.851,-112.657,173.775,38.105,157.242
C03076=1055.841,358.603,-112.619,173.771,38.100,157.241
C03077=1055.834,358.356,-112.582,173.766,38.095,157.240
C03078=1055.826,358.109,-112.544,173.761,38.090,157.238
C03079=1055.819,357.863,-112.506,173.757,38.085,157.237
C03080=1055.812,357.616,-112.468,173.752,38.079,157.236
C03081=1055.805,357.369,-112.431,173.747,38.074,157.235
C03082=1055.798,357.122,-112.394,173.743,38.069,157.233
C03083=1055.790,356.875,-112.356,173.738,38.064,157.232
C03084=1055.783,356.628,-112.319,173.733,38.059,157.231
C03085=1055.776,356.381,-112.281,173.729,38.054,157.229
C03086=1055.769,356.133,-112.244,173.724,38.049,157.228
C03087=1055.761,355.886,-112.206,173.719,38.043,157.227
C03088=1055.754,355.639,-112.169,173.715,38.038,157.226
C03089=1055.748,355.392,-112.130,173.710,38.033,157.224
C03090=1055.741,355.145,-112.093,173.706,38.028,157.223
C03091=1055.734,354.898,-112.056,173.701,38.023,157.222
C03092=1055.727,354.650,-112.019,173.696,38.018,157.221
C03093=1055.720,354.403,-111.981,173.692,38.013,157.219
C03094=1055.712,354.156,-111.944,173.687,38.008,157.218
C03095=1055.705,353.909,-111.906,173.683,38.003,157.217
C03096=1055.699,353.663,-111.869,173.678,37.998,157.216
C03097=1055.692,353.415,-111.832,173.674,37.993,157.214
C03098=1055.684,353.168,-111.795,173.669,37.988,157.213
C03099=1055.677,352.920,-111.757,173.664,37.983,157.212
C03100=1055.670,352.674,-111.720,173.660,37.978,157.211
C03101=1055.663,352.427,-111.684,173.655,37.973,157.209
C03102=1055.656,352.179,-111.646,173.651,37.968,157.208
C03103=1055.649,351.933,-111.609,173.646,37.963,157.207
C03104=1055.642,351.685,-111.572,173.642,37.958,157.206
C03105=1055.635,351.438,-111.535,173.637,37.953,157.204
C03106=1055.628,351.191,-111.499,173.633,37.948,157.203
C03107=1055.621,350.944,-111.461,173.628,37.943,157.202
C03108=1055.614,350.696,-111.424,173.624,37.938,157.201
C03109=1055.606,350.449,-111.387,173.619,37.933,157.200
C03110=1055.600,350.202,-111.351,173.615,37.928,157.198
C03111=1055.593,349.955,-111.313,173.610,37.924,157.197
C03112=1055.586,349.707,-111.276,173.606,37.919,157.196
C03113=1055.578,349.461,-111.240,173.601,37.914,157.195
C03114=1055.571,349.214,-111.203,173.597,37.909,157.194
C03115=1055.564,348.966,-111.166,173.592,37.904,157.192
C03116=1055.558,348.719,-111.129,173.588,37.899,157.191
C03117=1055.550,348.472,-111.093,173.584,37.895,157.190
C03118=1055.544,348.225,-111.056,173.580,37.890,157.189
C03119=1055.537,347.977,-111.020,173.575,37.885,157.188
C03120=1055.530,347.731,-110.982,173.571,37.880,157.186
C03121=1055.523,347.483,-110.946,173.566,37.875,157.185
C03122=1055.516,347.235,-110.909,173.562,37.870,157.184
C03123=1055.509,346.988,-110.873,173.557,37.866,157.183
C03124=1055.502,346.741,-110.837,173.553,37.861,157.182
C03125=1055.495,346.479,-110.797,173.548,37.856,157.181
C03126=1055.487,346.216,-110.758,173.544,37.851,157.179
C03127=1055.479,345.953,-110.720,173.539,37.846,157.178
C03128=1055.473,345.690,-110.681,173.534,37.841,157.177
C03129=1055.465,345.443,-110.645,173.530,37.836,157.176
C03130=1055.459,345.196,-110.609,173.526,37.831,157.175
C03131=1055.452,344.948,-110.572,173.522,37.826,157.173
C03132=1055.445,344.701,-110.536,173.518,37.822,157.172
C03133=1055.438,344.454,-110.499,173.513,37.817,157.171
C03134=1055.431,344.207,-110.463,173.509,37.813,157.170
C03135=1055.424,343.960,-110.427,173.505,37.808,157.169
C03136=1055.417,343.712,-110.391,173.500,37.803,157.168
C03137=1055.410,343.465,-110.354,173.496,37.799,157.167
C03138=1055.404,343.218,-110.317,173.492,37.794,157.165
C03139=1055.396,342.971,-110.281,173.488,37.789,157.164
C03140=1055.390,342.723,-110.245,173.484,37.784,157.163
C03141=1055.383,342.476,-110.209,173.479,37.780,157.162
C03142=1055.376,342.229,-110.174,173.475,37.775,157.161
C03143=1055.369,341.981,-110.137,173.471,37.771,157.160
C03144=1055.362,341.734,-110.102,173.466,37.766,157.159
C03145=1055.354,341.486,-110.065,173.462,37.761,157.157
C03146=1055.348,341.239,-110.029,173.458,37.757,157.156
C03147=1055.341,340.992,-109.994,173.454,37.752,157.155
C03148=1055.334,340.744,-109.957,173.450,37.748,157.154
C03149=1055.327,340.498,-109.921,173.446,37.744,157.153
C03150=1055.320,340.250,-109.886,173.441,37.739,157.152
C03151=1055.313,340.002,-109.849,173.437,37.734,157.151
C03152=1055.307,339.755,-109.814,173.433,37.730,157.150
C03153=1055.300,339.508,-109.778,173.429,37.725,157.149
C03154=1055.293,339.261,-109.741,173.425,37.721,157.148
C03155=1055.286,339.013,-109.706,173.421,37.716,157.146
C03156=1055.279,338.766,-109.670,173.416,37.712,157.145
C03157=1055.273,338.519,-109.635,173.412,37.707,157.144
C03158=1055.265,338.271,-109.599,173.408,37.702,157.143
C03159=1055.258,338.024,-109.563,173.405,37.698,157.142
C03160=1055.252,337.776,-109.528,173.400,37.693,157.141
C03161=1055.245,337.530,-109.492,173.396,37.689,157.140
C03162=1055.238,337.282,-109.457,173.392,37.684,157.139
C03163=1055.232,337.034,-109.420,173.388,37.680,157.138
C03164=1055.225,336.787,-109.385,173.383,37.675,157.137
C03165=1055.218,336.540,-109.350,173.380,37.671,157.136
C03166=1055.211,336.292,-109.314,173.376,37.666,157.134
C03167=1055.204,336.045,-109.278,173.372,37.662,157.134
C03168=1055.198,335.797,-109.243,173.367,37.658,157.132
C03169=1055.191,335.550,-109.207,173.363,37.654,157.131
C03170=1055.184,335.302,-109.172,173.360,37.649,157.130
C03171=1055.177,335.055,-109.137,173.356,37.645,157.129
C03172=1055.170,334.808,-109.101,173.351,37.640,157.128
C03173=1055.163,334.560,-109.066,173.347,37.636,157.127
C03174=1055.156,334.313,-109.031,173.344,37.632,157.126
C03175=1055.149,334.066,-108.996,173.340,37.627,157.125
C03176=1055.142,333.818,-108.960,173.335,37.623,157.124
C03177=1055.136,333.571,-108.925,173.331,37.618,157.123
C03178=1055.129,333.323,-108.890,173.327,37.614,157.122
C03179=1055.123,333.076,-108.854,173.324,37.610,157.121
C03180=1055.116,332.828,-108.819,173.320,37.605,157.120
C03181=1055.108,332.561,-108.781,173.315,37.601,157.119
C03182=1055.101,332.295,-108.744,173.311,37.596,157.118
C03183=1055.094,332.028,-108.705,173.306,37.591,157.116
C03184=1055.086,331.761,-108.668,173.303,37.587,157.115
C03185=1055.080,331.514,-108.633,173.299,37.582,157.114
C03186=1055.073,331.267,-108.597,173.295,37.578,157.113
C03187=1055.066,331.019,-108.562,173.290,37.574,157.112
C03188=1055.060,330.771,-108.528,173.286,37.569,157.111
C03189=1055.053,330.524,-108.492,173.283,37.565,157.110
C03190=1055.047,330.276,-108.457,173.279,37.561,157.109
C03191=1055.039,330.029,-108.422,173.275,37.556,157.108
C03192=1055.032,329.782,-108.387,173.271,37.553,157.107
C03193=1055.025,329.533,-108.353,173.268,37.548,157.106
C03194=1055.018,329.286,-108.318,173.263,37.544,157.105
C03195=1055.011,329.039,-108.283,173.259,37.540,157.104
C03196=1055.005,328.791,-108.248,173.255,37.536,157.103
C03197=1054.998,328.543,-108.213,173.252,37.532,157.102
C03198=1054.990,328.296,-108.179,173.248,37.527,157.101
C03199=1054.984,328.048,-108.144,173.244,37.523,157.100
C03200=1054.976,327.801,-108.110,173.241,37.519,157.099
C03201=1054.970,327.553,-108.075,173.236,37.515,157.098
C03202=1054.963,327.306,-108.040,173.232,37.511,157.097
C03203=1054.956,327.058,-108.006,173.228,37.507,157.096
C03204=1054.950,326.812,-107.972,173.225,37.502,157.095
C03205=1054.943,326.564,-107.937,173.221,37.498,157.094
C03206=1054.936,326.317,-107.903,173.217,37.495,157.093
C03207=1054.929,326.069,-107.868,173.214,37.490,157.092
C03208=1054.923,325.821,-107.833,173.210,37.486,157.091
C03209=1054.915,325.573,-107.799,173.206,37.482,157.091
C03210=1054.909,325.326,-107.764,173.201,37.478,157.089
C03211=1054.901,325.078,-107.730,173.198,37.474,157.089
C03212=1054.895,324.830,-107.696,173.194,37.470,157.088
C03213=1054.888,324.583,-107.661,173.190,37.465,157.087
C03214=1054.882,324.336,-107.627,173.187,37.461,157.086
C03215=1054.875,324.088,-107.593,173.183,37.457,157.085
C03216=1054.868,323.841,-107.558,173.179,37.453,157.084
C03217=1054.861,323.593,-107.524,173.175,37.449,157.083
C03218=1054.855,323.345,-107.490,173.172,37.445,157.082
C03219=1054.848,323.099,-107.455,173.168,37.441,157.081
C03220=1054.841,322.851,-107.421,173.164,37.437,157.080
C03221=1054.834,322.603,-107.387,173.161,37.433,157.079
C03222=1054.828,322.355,-107.353,173.157,37.428,157.078
C03223=1054.821,322.107,-107.318,173.153,37.425,157.077
C03224=1054.814,321.861,-107.284,173.150,37.421,157.076
C03225=1054.808,321.613,-107.250,173.146,37.417,157.075
C03226=1054.801,321.365,-107.216,173.142,37.413,157.074
C03227=1054.795,321.118,-107.182,173.138,37.408,157.073
C03228=1054.788,320.870,-107.148,173.135,37.404,157.072
C03229=1054.781,320.622,-107.114,173.131,37.400,157.071
C03230=1054.775,320.374,-107.079,173.127,37.396,157.070
C03231=1054.768,320.127,-107.046,173.124,37.392,157.069
C03232=1054.762,319.879,-107.011,173.120,37.388,157.068
C03233=1054.754,319.632,-106.977,173.116,37.384,157.068
C03234=1054.749,319.384,-106.943,173.113,37.380,157.067
C03235=1054.741,319.137,-106.910,173.109,37.376,157.066
C03236=1054.735,318.889,-106.876,173.105,37.372,157.065
C03237=1054.728,318.617,-106.837,173.102,37.367,157.064
C03238=1054.720,318.345,-106.801,173.097,37.363,157.063
C03239=1054.713,318.073,-106.763,173.093,37.359,157.062
C03240=1054.706,317.801,-106.726,173.089,37.354,157.061
C03241=1054.700,317.553,-106.692,173.086,37.350,157.060
C03242=1054.693,317.306,-106.658,173.082,37.346,157.059
C03243=1054.687,317.058,-106.624,173.078,37.342,157.058
C03244=1054.680,316.810,-106.591,173.075,37.338,157.057
C03245=1054.674,316.562,-106.557,173.071,37.334,157.056
C03246=1054.667,316.315,-106.523,173.067,37.330,157.055
C03247=1054.661,316.067,-106.489,173.065,37.326,157.054
C03248=1054.654,315.820,-106.455,173.061,37.322,157.053
C03249=1054.648,315.572,-106.422,173.058,37.318,157.052
C03250=1054.641,315.324,-106.388,173.054,37.314,157.051
C03251=1054.635,315.077,-106.354,173.050,37.310,157.050
C03252=1054.628,314.829,-106.320,173.047,37.307,157.049
C03253=1054.622,314.581,-106.286,173.043,37.303,157.049
C03254=1054.616,314.334,-106.253,173.039,37.299,157.048
C03255=1054.609,314.087,-106.219,173.036,37.295,157.047
C03256=1054.603,313.839,-106.186,173.033,37.291,157.046
C03257=1054.596,313.591,-106.152,173.029,37.287,157.045
C03258=1054.590,313.344,-106.118,173.026,37.283,157.044
C03259=1054.583,313.096,-106.085,173.022,37.279,157.043
C03260=1054.576,312.849,-106.051,173.018,37.275,157.042
C03261=1054.570,312.600,-106.018,173.015,37.271,157.041
C03262=1054.563,312.353,-105.985,173.011,37.267,157.040
C03263=1054.556,312.105,-105.952,173.007,37.263,157.039
C03264=1054.549,311.858,-105.918,173.004,37.260,157.039
C03265=1054.543,311.610,-105.885,173.000,37.256,157.038
C03266=1054.536,311.362,-105.852,172.998,37.252,157.037
C03267=1054.529,311.114,-105.819,172.994,37.248,157.036
C03268=1054.522,310.867,-105.786,172.990,37.244,157.035
C03269=1054.515,310.619,-105.753,172.987,37.240,157.034
C03270=1054.509,310.372,-105.720,172.983,37.237,157.033
C03271=1054.502,310.124,-105.687,172.980,37.233,157.032
C03272=1054.495,309.876,-105.654,172.976,37.229,157.032
C03273=1054.489,309.629,-105.621,172.972,37.226,157.031
C03274=1054.482,309.381,-105.587,172.970,37.222,157.030
C03275=1054.476,309.133,-105.555,172.966,37.218,157.029
C03276=1054.469,308.885,-105.522,172.963,37.214,157.028
C03277=1054.462,308.638,-105.488,172.959,37.210,157.027
C03278=1054.456,308.390,-105.455,172.955,37.207,157.026
C03279=1054.449,308.142,-105.422,172.952,37.203,157.025
C03280=1054.442,307.895,-105.390,172.949,37.199,157.025
C03281=1054.436,307.647,-105.357,172.946,37.195,157.024
C03282=1054.428,307.399,-105.324,172.942,37.191,157.023
C03283=1054.422,307.152,-105.291,172.938,37.188,157.022
C03284=1054.416,306.904,-105.258,172.935,37.184,157.021
C03285=1054.409,306.656,-105.225,172.931,37.180,157.020
C03286=1054.403,306.408,-105.192,172.929,37.176,157.019
C03287=1054.396,306.161,-105.159,172.925,37.172,157.019
C03288=1054.389,305.914,-105.127,172.921,37.169,157.018
C03289=1054.382,305.665,-105.094,172.918,37.165,157.017
C03290=1054.376,305.418,-105.061,172.914,37.162,157.016
C03291=1054.370,305.170,-105.029,172.912,37.158,157.015
C03292=1054.363,304.922,-104.996,172.908,37.154,157.014
C03293=1054.356,304.655,-104.960,172.904,37.150,157.013
C03294=1054.349,304.387,-104.925,172.901,37.146,157.012
C03295=1054.342,304.118,-104.890,172.897,37.142,157.011
C03296=1054.335,303.851,-104.854,172.893,37.138,157.011
C03297=1054.329,303.603,-104.821,172.890,37.134,157.010
C03298=1054.321,303.355,-104.789,172.886,37.130,157.009
C03299=1054.315,303.108,-104.756,172.884,37.127,157.008
C03300=1054.309,302.859,-104.724,172.880,37.123,157.007
C03301=1054.303,302.612,-104.691,172.877,37.119,157.006
C03302=1054.296,302.364,-104.658,172.874,37.115,157.005
C03303=1054.290,302.117,-104.626,172.870,37.112,157.005
C03304=1054.283,301.869,-104.593,172.867,37.108,157.004
C03305=1054.276,301.621,-104.560,172.863,37.104,157.003
C03306=1054.270,301.373,-104.528,172.861,37.100,157.002
C03307=1054.264,301.125,-104.495,172.857,37.097,157.001
C03308=1054.257,300.878,-104.463,172.854,37.093,157.000
C03309=1054.250,300.630,-104.431,172.851,37.089,157.000
C03310=1054.244,300.382,-104.399,172.847,37.085,156.999
C03311=1054.238,300.134,-104.366,172.844,37.082,156.998
C03312=1054.232,299.887,-104.333,172.840,37.078,156.997
C03313=1054.226,299.639,-104.300,172.838,37.074,156.996
C03314=1054.219,299.391,-104.269,172.834,37.070,156.995
C03315=1054.213,299.144,-104.236,172.831,37.067,156.995
C03316=1054.207,298.896,-104.204,172.828,37.063,156.994
C03317=1054.200,298.648,-104.171,172.824,37.059,156.993
C03318=1054.194,298.400,-104.139,172.821,37.055,156.992
C03319=1054.187,298.152,-104.107,172.818,37.052,156.991
C03320=1054.181,297.905,-104.074,172.815,37.048,156.990
C03321=1054.175,297.657,-104.042,172.811,37.044,156.989
C03322=1054.169,297.409,-104.010,172.809,37.040,156.989
C03323=1054.162,297.162,-103.978,172.805,37.037,156.988
C03324=1054.156,296.914,-103.946,172.801,37.033,156.987
C03325=1054.149,296.666,-103.913,172.799,37.029,156.986
C03326=1054.143,296.418,-103.881,172.795,37.026,156.985
C03327=1054.137,296.170,-103.849,172.793,37.022,156.984
C03328=1054.130,295.922,-103.817,172.789,37.019,156.984
C03329=1054.124,295.674,-103.785,172.786,37.015,156.983
C03330=1054.117,295.427,-103.752,172.783,37.012,156.982
C03331=1054.111,295.179,-103.721,172.780,37.008,156.981
C03332=1054.105,294.931,-103.689,172.776,37.004,156.980
C03333=1054.098,294.683,-103.657,172.774,37.001,156.980
C03334=1054.092,294.435,-103.625,172.770,36.997,156.979
C03335=1054.085,294.187,-103.593,172.766,36.993,156.978
C03336=1054.078,293.940,-103.561,172.764,36.990,156.977
C03337=1054.072,293.692,-103.529,172.760,36.986,156.976
C03338=1054.065,293.444,-103.498,172.758,36.983,156.976
C03339=1054.058,293.196,-103.466,172.754,36.979,156.975
C03340=1054.052,292.948,-103.434,172.751,36.975,156.974
C03341=1054.045,292.700,-103.402,172.748,36.972,156.973
C03342=1054.039,292.453,-103.371,172.745,36.968,156.972
C03343=1054.033,292.204,-103.339,172.742,36.965,156.972
C03344=1054.026,291.956,-103.307,172.739,36.961,156.971
C03345=1054.020,291.708,-103.275,172.735,36.957,156.970
C03346=1054.013,291.460,-103.244,172.733,36.954,156.969
C03347=1054.007,291.212,-103.212,172.729,36.950,156.968
C03348=1054.000,290.965,-103.180,172.727,36.947,156.968
C03349=1053.993,290.713,-103.149,172.723,36.943,156.967
C03350=1053.987,290.461,-103.116,172.719,36.939,156.966
C03351=1053.981,290.209,-103.084,172.717,36.936,156.965
C03352=1053.974,289.957,-103.052,172.713,36.932,156.964
C03353=1053.967,289.709,-103.020,172.711,36.928,156.963
C03354=1053.961,289.461,-102.989,172.707,36.925,156.963
C03355=1053.955,289.213,-102.957,172.704,36.921,156.962
C03356=1053.948,288.965,-102.925,172.701,36.918,156.961
C03357=1053.942,288.718,-102.894,172.698,36.915,156.960
C03358=1053.936,288.470,-102.862,172.695,36.911,156.960
C03359=1053.929,288.222,-102.831,172.692,36.908,156.959
C03360=1053.923,287.973,-102.800,172.689,36.904,156.958
C03361=1053.916,287.725,-102.769,172.686,36.900,156.957
C03362=1053.909,287.477,-102.737,172.683,36.897,156.956
C03363=1053.903,287.230,-102.706,172.680,36.893,156.956
C03364=1053.896,286.982,-102.675,172.676,36.890,156.955
C03365=1053.890,286.734,-102.643,172.674,36.886,156.954
C03366=1053.883,286.486,-102.613,172.670,36.883,156.953
C03367=1053.877,286.238,-102.581,172.668,36.879,156.952
C03368=1053.870,285.990,-102.550,172.664,36.876,156.952
C03369=1053.864,285.742,-102.518,172.662,36.872,156.951
C03370=1053.858,285.494,-102.487,172.658,36.869,156.950
C03371=1053.851,285.246,-102.456,172.656,36.865,156.949
C03372=1053.845,284.998,-102.425,172.652,36.862,156.949
C03373=1053.839,284.750,-102.394,172.650,36.858,156.948
C03374=1053.832,284.502,-102.363,172.646,36.855,156.947
C03375=1053.825,284.254,-102.331,172.644,36.851,156.946
C03376=1053.819,284.006,-102.301,172.640,36.848,156.946
C03377=1053.813,283.759,-102.270,172.638,36.844,156.945
C03378=1053.806,283.511,-102.238,172.634,36.841,156.944
C03379=1053.800,283.262,-102.207,172.632,36.837,156.943
C03380=1053.793,283.014,-102.176,172.628,36.834,156.942
C03381=1053.787,282.767,-102.146,172.626,36.830,156.942
C03382=1053.780,282.519,-102.114,172.622,36.827,156.941
C03383=1053.774,282.271,-102.083,172.620,36.823,156.940
C03384=1053.768,282.023,-102.052,172.616,36.820,156.939
C03385=1053.761,281.775,-102.021,172.614,36.816,156.939
C03386=1053.755,281.527,-101.990,172.611,36.813,156.938
C03387=1053.749,281.279,-101.959,172.608,36.809,156.937
C03388=1053.742,281.031,-101.928,172.605,36.805,156.936
C03389=1053.735,280.783,-101.897,172.602,36.802,156.935
C03390=1053.730,280.535,-101.867,172.599,36.798,156.935
C03391=1053.723,280.287,-101.835,172.596,36.795,156.934
C03392=1053.716,280.039,-101.805,172.593,36.791,156.933
C03393=1053.711,279.791,-101.774,172.590,36.788,156.932
C03394=1053.704,279.543,-101.743,172.587,36.784,156.932
C03395=1053.697,279.294,-101.712,172.585,36.782,156.931
C03396=1053.691,279.047,-101.682,172.581,36.778,156.930
C03397=1053.684,278.799,-101.651,172.579,36.775,156.929
C03398=1053.678,278.551,-101.621,172.575,36.771,156.929
C03399=1053.672,278.303,-101.590,172.573,36.768,156.928
C03400=1053.665,278.055,-101.558,172.569,36.764,156.927
C03401=1053.659,277.810,-101.528,172.567,36.761,156.926
C03402=1053.653,277.566,-101.498,172.564,36.757,156.926
C03403=1053.646,277.322,-101.469,172.561,36.754,156.925
C03404=1053.640,277.077,-101.439,172.559,36.751,156.924
C03405=1053.634,276.832,-101.408,172.556,36.747,156.923
C03406=1053.627,276.588,-101.378,172.553,36.744,156.923
C03407=1053.621,276.343,-101.348,172.550,36.740,156.922
C03408=1053.615,276.100,-101.318,172.547,36.737,156.921
C03409=1053.608,275.851,-101.287,172.544,36.733,156.920
C03410=1053.602,275.603,-101.257,172.542,36.730,156.920
C03411=1053.595,275.355,-101.227,172.538,36.727,156.919
C03412=1053.589,275.107,-101.196,172.536,36.723,156.918
C03413=1053.583,274.859,-101.165,172.533,36.720,156.917
C03414=1053.576,274.611,-101.135,172.530,36.716,156.917
C03415=1053.570,274.363,-101.105,172.527,36.713,156.916
C03416=1053.564,274.114,-101.074,172.524,36.709,156.915
C03417=1053.557,273.867,-101.045,172.521,36.706,156.914
C03418=1053.551,273.618,-101.014,172.519,36.702,156.914
C03419=1053.545,273.370,-100.983,172.516,36.699,156.913
C03420=1053.538,273.122,-100.953,172.513,36.696,156.912
C03421=1053.532,272.874,-100.923,172.511,36.692,156.911
C03422=1053.525,272.626,-100.892,172.507,36.689,156.911
C03423=1053.519,272.378,-100.863,172.505,36.685,156.910
C03424=1053.512,272.130,-100.832,172.502,36.682,156.909
C03425=1053.506,271.882,-100.802,172.499,36.678,156.908
C03426=1053.499,271.634,-100.771,172.496,36.675,156.908
C03427=1053.494,271.386,-100.741,172.494,36.672,156.907
C03428=1053.487,271.138,-100.711,172.490,36.668,156.906
C03429=1053.481,270.890,-100.680,172.488,36.665,156.905
C03430=1053.474,270.642,-100.650,172.485,36.661,156.905
C03431=1053.468,270.393,-100.621,172.482,36.658,156.904
C03432=1053.461,270.146,-100.591,172.480,36.655,156.903
C03433=1053.455,269.897,-100.560,172.477,36.651,156.902
C03434=1053.448,269.650,-100.531,172.474,36.648,156.902
C03435=1053.442,269.401,-100.500,172.471,36.644,156.901
C03436=1053.436,269.153,-100.471,172.469,36.641,156.900
C03437=1053.429,268.905,-100.440,172.465,36.638,156.900
C03438=1053.423,268.657,-100.410,172.463,36.634,156.899
C03439=1053.416,268.410,-100.381,172.460,36.631,156.898
C03440=1053.410,268.160,-100.351,172.457,36.627,156.897
C03441=1053.404,267.913,-100.321,172.454,36.624,156.897
C03442=1053.397,267.664,-100.290,172.452,36.621,156.896
C03443=1053.391,267.416,-100.261,172.450,36.617,156.895
C03444=1053.384,267.169,-100.231,172.446,36.614,156.894
C03445=1053.378,266.920,-100.201,172.444,36.610,156.894
C03446=1053.372,266.672,-100.171,172.441,36.607,156.893
C03447=1053.365,266.424,-100.141,172.438,36.604,156.892
C03448=1053.359,266.175,-100.112,172.435,36.600,156.891
C03449=1053.353,265.928,-100.082,172.433,36.597,156.891
C03450=1053.346,265.679,-100.053,172.430,36.593,156.890
C03451=1053.340,265.431,-100.022,172.427,36.590,156.889
C03452=1053.334,265.183,-99.993,172.425,36.587,156.889
C03453=1053.326,264.935,-99.963,172.422,36.583,156.888
C03454=1053.321,264.687,-99.933,172.420,36.580,156.887
C03455=1053.314,264.439,-99.904,172.416,36.577,156.886
C03456=1053.308,264.190,-99.874,172.414,36.573,156.886
C03457=1053.302,263.948,-99.845,172.411,36.570,156.885
C03458=1053.296,263.706,-99.816,172.409,36.566,156.884
C03459=1053.289,263.463,-99.787,172.406,36.563,156.883
C03460=1053.283,263.221,-99.758,172.403,36.560,156.883
C03461=1053.277,262.979,-99.729,172.401,36.556,156.882
C03462=1053.270,262.736,-99.700,172.398,36.553,156.881
C03463=1053.264,262.494,-99.671,172.396,36.550,156.881
C03464=1053.258,262.251,-99.643,172.393,36.547,156.880
C03465=1053.251,262.003,-99.613,172.390,36.543,156.879
C03466=1053.245,261.755,-99.584,172.388,36.540,156.879
C03467=1053.238,261.506,-99.555,172.385,36.537,156.878
C03468=1053.232,261.258,-99.526,172.383,36.533,156.877
C03469=1053.225,261.011,-99.496,172.379,36.530,156.876
C03470=1053.218,260.762,-99.467,172.377,36.527,156.876
C03471=1053.212,260.514,-99.437,172.374,36.524,156.875
C03472=1053.206,260.266,-99.408,172.372,36.520,156.874
C03473=1053.199,260.017,-99.378,172.369,36.517,156.874
C03474=1053.192,259.769,-99.349,172.366,36.514,156.873
C03475=1053.186,259.521,-99.320,172.364,36.510,156.872
C03476=1053.180,259.273,-99.291,172.361,36.507,156.871
C03477=1053.173,259.024,-99.262,172.359,36.504,156.871
C03478=1053.167,258.776,-99.233,172.355,36.500,156.870
C03479=1053.160,258.529,-99.203,172.353,36.497,156.869
C03480=1053.154,258.280,-99.174,172.351,36.494,156.869
C03481=1053.147,258.032,-99.145,172.348,36.490,156.868
C03482=1053.141,257.784,-99.116,172.346,36.487,156.867
C03483=1053.135,257.535,-99.086,172.342,36.484,156.866
C03484=1053.128,257.287,-99.057,172.340,36.480,156.866
C03485=1053.121,257.039,-99.029,172.337,36.477,156.865
C03486=1053.115,256.791,-99.000,172.335,36.474,156.864
C03487=1053.108,256.542,-98.971,172.333,36.470,156.864
C03488=1053.102,256.294,-98.942,172.330,36.467,156.863
C03489=1053.096,256.046,-98.912,172.327,36.464,156.862
C03490=1053.089,255.797,-98.883,172.324,36.460,156.861
C03491=1053.083,255.549,-98.854,172.322,36.457,156.861
C03492=1053.076,255.301,-98.825,172.320,36.454,156.860
C03493=1053.070,255.053,-98.796,172.317,36.450,156.859
C03494=1053.064,254.805,-98.767,172.315,36.447,156.859
C03495=1053.058,254.557,-98.738,172.312,36.444,156.858
C03496=1053.051,254.309,-98.709,172.309,36.440,156.857
C03497=1053.045,254.060,-98.679,172.306,36.437,156.856
C03498=1053.038,253.812,-98.651,172.304,36.434,156.856
C03499=1053.031,253.564,-98.622,172.302,36.430,156.855
C03500=1053.025,253.315,-98.594,172.299,36.427,156.854
C03501=1053.019,253.067,-98.565,172.297,36.424,156.854
C03502=1053.013,252.819,-98.536,172.294,36.420,156.853
C03503=1053.007,252.571,-98.506,172.292,36.416,156.852
C03504=1053.000,252.323,-98.477,172.288,36.413,156.851
C03505=1052.994,252.074,-98.448,172.286,36.410,156.851
C03506=1052.988,251.826,-98.420,172.284,36.406,156.850
C03507=1052.981,251.578,-98.392,172.281,36.403,156.849
C03508=1052.975,251.330,-98.363,172.279,36.400,156.849
C03509=1052.968,251.081,-98.333,172.276,36.396,156.848
C03510=1052.962,250.833,-98.304,172.274,36.393,156.847
C03511=1052.956,250.584,-98.276,172.272,36.389,156.846
C03512=1052.950,250.336,-98.247,172.269,36.386,156.846
C03513=1052.944,250.092,-98.219,172.267,36.383,156.845
C03514=1052.937,249.850,-98.190,172.264,36.379,156.844
C03515=1052.932,249.606,-98.163,172.262,36.376,156.844
C03516=1052.925,249.363,-98.134,172.260,36.373,156.843
C03517=1052.919,249.119,-98.106,172.257,36.370,156.842
C03518=1052.913,248.876,-98.078,172.255,36.366,156.842
C03519=1052.907,248.633,-98.050,172.252,36.363,156.841
C03520=1052.901,248.390,-98.022,172.250,36.360,156.840
C03521=1052.895,248.141,-97.993,172.247,36.356,156.839
C03522=1052.888,247.893,-97.964,172.244,36.353,156.839
C03523=1052.882,247.645,-97.935,172.242,36.349,156.838
C03524=1052.876,247.396,-97.907,172.239,36.346,156.837
C03525=1052.869,247.148,-97.879,172.237,36.342,156.837
C03526=1052.863,246.899,-97.850,172.234,36.339,156.836
C03527=1052.857,246.651,-97.821,172.232,36.335,156.835
C03528=1052.851,246.403,-97.792,172.230,36.332,156.834
C03529=1052.845,246.155,-97.764,172.227,36.329,156.834
C03530=1052.839,245.907,-97.735,172.225,36.325,156.833
C03531=1052.833,245.659,-97.707,172.222,36.322,156.832
C03532=1052.827,245.410,-97.679,172.220,36.319,156.832
C03533=1052.820,245.162,-97.651,172.218,36.315,156.831
C03534=1052.814,244.913,-97.622,172.215,36.312,156.830
C03535=1052.807,244.665,-97.593,172.213,36.309,156.829
C03536=1052.801,244.417,-97.566,172.210,36.305,156.829
C03537=1052.794,244.169,-97.537,172.208,36.302,156.828
C03538=1052.788,243.920,-97.509,172.206,36.299,156.827
C03539=1052.782,243.671,-97.480,172.203,36.295,156.827
C03540=1052.776,243.423,-97.451,172.201,36.291,156.826
C03541=1052.769,243.175,-97.424,172.198,36.288,156.825
C03542=1052.763,242.926,-97.395,172.196,36.285,156.824
C03543=1052.757,242.679,-97.367,172.194,36.281,156.824
C03544=1052.751,242.430,-97.339,172.191,36.278,156.823
C03545=1052.744,242.182,-97.311,172.189,36.275,156.822
C03546=1052.738,241.934,-97.282,172.186,36.271,156.822
C03547=1052.732,241.685,-97.254,172.184,36.268,156.821
C03548=1052.725,241.436,-97.226,172.182,36.265,156.820
C03549=1052.718,241.188,-97.198,172.179,36.261,156.819
C03550=1052.712,240.940,-97.169,172.177,36.258,156.819
C03551=1052.705,240.691,-97.142,172.175,36.255,156.818
C03552=1052.699,240.444,-97.114,172.172,36.251,156.817
C03553=1052.693,240.195,-97.086,172.170,36.248,156.817
C03554=1052.687,239.946,-97.058,172.167,36.245,156.816
C03555=1052.680,239.698,-97.030,172.165,36.241,156.815
C03556=1052.674,239.450,-97.001,172.163,36.238,156.815
C03557=1052.667,239.201,-96.974,172.160,36.234,156.814
C03558=1052.660,238.953,-96.946,172.158,36.231,156.813
C03559=1052.655,238.705,-96.918,172.155,36.228,156.812
C03560=1052.648,238.457,-96.890,172.153,36.224,156.812
C03561=1052.642,238.208,-96.863,172.151,36.221,156.811
C03562=1052.636,237.959,-96.834,172.148,36.218,156.810
C03563=1052.629,237.711,-96.807,172.146,36.214,156.810
C03564=1052.622,237.462,-96.779,172.144,36.211,156.809
C03565=1052.617,237.214,-96.751,172.142,36.208,156.808
C03566=1052.610,236.966,-96.723,172.140,36.204,156.808
C03567=1052.604,236.717,-96.695,172.137,36.201,156.807
C03568=1052.597,236.469,-96.668,172.135,36.198,156.806
C03569=1052.591,236.223,-96.640,172.133,36.194,156.805
C03570=1052.585,235.977,-96.613,172.130,36.190,156.805
C03571=1052.579,235.731,-96.584,172.128,36.187,156.804
C03572=1052.572,235.484,-96.557,172.125,36.184,156.803
C03573=1052.566,235.238,-96.529,172.123,36.181,156.803
C03574=1052.559,234.992,-96.502,172.121,36.177,156.802
C03575=1052.553,234.745,-96.474,172.118,36.174,156.801
C03576=1052.547,234.499,-96.447,172.117,36.171,156.801
C03577=1052.541,234.250,-96.419,172.114,36.167,156.800
C03578=1052.535,234.001,-96.392,172.112,36.164,156.799
C03579=1052.528,233.754,-96.365,172.110,36.161,156.798
C03580=1052.522,233.505,-96.337,172.107,36.157,156.798
C03581=1052.516,233.256,-96.308,172.105,36.153,156.797
C03582=1052.509,233.008,-96.281,172.103,36.150,156.796
C03583=1052.503,232.760,-96.253,172.100,36.147,156.796
C03584=1052.497,232.511,-96.226,172.098,36.143,156.795
C03585=1052.490,232.263,-96.199,172.096,36.140,156.794
C03586=1052.485,232.015,-96.171,172.094,36.137,156.794
C03587=1052.478,231.766,-96.143,172.092,36.133,156.793
C03588=1052.471,231.518,-96.115,172.089,36.130,156.792
C03589=1052.465,231.269,-96.088,172.087,36.127,156.791
C03590=1052.459,231.021,-96.061,172.085,36.123,156.791
C03591=1052.452,230.772,-96.033,172.082,36.119,156.790
C03592=1052.446,230.523,-96.006,172.080,36.116,156.789
C03593=1052.440,230.276,-95.979,172.078,36.113,156.789
C03594=1052.433,230.027,-95.951,172.076,36.109,156.788
C03595=1052.427,229.778,-95.923,172.074,36.106,156.787
C03596=1052.421,229.530,-95.896,172.071,36.103,156.787
C03597=1052.415,229.282,-95.868,172.069,36.099,156.786
C03598=1052.409,229.033,-95.842,172.066,36.096,156.785
C03599=1052.402,228.785,-95.814,172.064,36.093,156.784
C03600=1052.396,228.536,-95.786,172.063,36.089,156.784
C03601=1052.388,228.288,-95.760,172.060,36.085,156.783
C03602=1052.382,228.040,-95.732,172.058,36.082,156.782
C03603=1052.376,227.791,-95.705,172.056,36.079,156.782
C03604=1052.369,227.542,-95.678,172.053,36.075,156.781
